C01819=1081.465,156.969,428.718,174.663,22.838,153.849
C01820=1081.471,157.219,428.696,174.666,22.840,153.849
C01821=1081.476,157.468,428.675,174.667,22.842,153.849
C01822=1081.482,157.716,428.654,174.670,22.844,153.849
C01823=1081.488,157.966,428.633,174.672,22.846,153.850
C01824=1081.493,158.215,428.611,174.674,22.848,153.850
C01825=1081.499,158.463,428.590,174.676,22.850,153.850
C01826=1081.505,158.713,428.569,174.678,22.852,153.850
C01827=1081.510,158.962,428.548,174.680,22.854,153.850
C01828=1081.517,159.241,428.524,174.683,22.857,153.850
C01829=1081.523,159.522,428.500,174.685,22.859,153.850
C01830=1081.529,159.801,428.476,174.687,22.861,153.850
C01831=1081.535,160.081,428.452,174.690,22.863,153.851
C01832=1081.541,160.330,428.430,174.692,22.866,153.851
C01833=1081.546,160.579,428.409,174.694,22.868,153.851
C01834=1081.552,160.829,428.388,174.697,22.870,153.851
C01835=1081.558,161.077,428.366,174.698,22.872,153.851
C01836=1081.564,161.327,428.345,174.701,22.874,153.851
C01837=1081.569,161.575,428.323,174.703,22.876,153.851
C01838=1081.574,161.824,428.302,174.705,22.879,153.851
C01839=1081.580,162.074,428.281,174.707,22.880,153.852
C01840=1081.585,162.323,428.259,174.709,22.883,153.852
C01841=1081.590,162.571,428.238,174.711,22.885,153.852
C01842=1081.596,162.821,428.215,174.714,22.887,153.852
C01843=1081.601,163.069,428.194,174.716,22.889,153.852
C01844=1081.608,163.318,428.172,174.718,22.891,153.852
C01845=1081.612,163.567,428.151,174.720,22.893,153.852
C01846=1081.619,163.816,428.129,174.722,22.895,153.853
C01847=1081.623,164.066,428.108,174.725,22.898,153.853
C01848=1081.629,164.314,428.086,174.727,22.900,153.853
C01849=1081.634,164.564,428.064,174.728,22.902,153.853
C01850=1081.640,164.812,428.043,174.731,22.904,153.853
C01851=1081.645,165.062,428.021,174.733,22.906,153.853
C01852=1081.651,165.310,427.999,174.735,22.908,153.853
C01853=1081.656,165.560,427.977,174.738,22.910,153.853
C01854=1081.662,165.808,427.956,174.739,22.912,153.854
C01855=1081.667,166.058,427.934,174.742,22.915,153.854
C01856=1081.673,166.306,427.912,174.744,22.917,153.854
C01857=1081.677,166.555,427.891,174.746,22.919,153.854
C01858=1081.684,166.804,427.869,174.749,22.921,153.854
C01859=1081.688,167.053,427.847,174.750,22.923,153.854
C01860=1081.695,167.302,427.825,174.752,22.925,153.854
C01861=1081.699,167.551,427.804,174.755,22.927,153.855
C01862=1081.706,167.800,427.782,174.757,22.930,153.855
C01863=1081.710,168.049,427.760,174.759,22.932,153.855
C01864=1081.716,168.298,427.738,174.761,22.933,153.855
C01865=1081.721,168.547,427.717,174.763,22.935,153.855
C01866=1081.728,168.796,427.694,174.766,22.938,153.855
C01867=1081.733,169.045,427.672,174.768,22.940,153.855
C01868=1081.739,169.294,427.651,174.770,22.942,153.855
C01869=1081.744,169.543,427.629,174.773,22.944,153.855
C01870=1081.749,169.792,427.607,174.774,22.946,153.856
C01871=1081.755,170.041,427.585,174.777,22.948,153.856
C01872=1081.760,170.290,427.563,174.779,22.950,153.856
C01873=1081.766,170.539,427.541,174.781,22.953,153.856
C01874=1081.771,170.788,427.519,174.784,22.954,153.856
C01875=1081.777,171.037,427.497,174.786,22.957,153.856
C01876=1081.783,171.286,427.475,174.788,22.959,153.856
C01877=1081.788,171.535,427.454,174.790,22.961,153.856
C01878=1081.794,171.784,427.431,174.792,22.963,153.856
C01879=1081.799,172.032,427.409,174.795,22.965,153.857
C01880=1081.805,172.282,427.387,174.797,22.967,153.857
C01881=1081.811,172.531,427.365,174.799,22.969,153.857
C01882=1081.816,172.779,427.343,174.801,22.971,153.857
C01883=1081.822,173.029,427.321,174.803,22.973,153.857
C01884=1081.827,173.278,427.299,174.806,22.975,153.857
C01885=1081.833,173.527,427.277,174.808,22.978,153.857
C01886=1081.839,173.776,427.254,174.810,22.979,153.857
C01887=1081.844,174.024,427.233,174.813,22.982,153.858
C01888=1081.850,174.274,427.211,174.815,22.984,153.858
C01889=1081.855,174.522,427.188,174.817,22.985,153.858
C01890=1081.861,174.771,427.167,174.819,22.988,153.858
C01891=1081.866,175.020,427.145,174.821,22.990,153.858
C01892=1081.873,175.300,427.119,174.824,22.992,153.858
C01893=1081.879,175.580,427.094,174.827,22.995,153.858
C01894=1081.886,175.859,427.069,174.829,22.997,153.858
C01895=1081.892,176.138,427.045,174.832,22.999,153.858
C01896=1081.897,176.387,427.023,174.834,23.001,153.859
C01897=1081.903,176.636,427.000,174.836,23.003,153.859
C01898=1081.909,176.885,426.978,174.839,23.005,153.859
C01899=1081.914,177.134,426.956,174.841,23.007,153.859
C01900=1081.920,177.383,426.933,174.843,23.009,153.859
C01901=1081.926,177.632,426.911,174.845,23.011,153.859
C01902=1081.932,177.881,426.889,174.847,23.013,153.859
C01903=1081.937,178.129,426.866,174.850,23.016,153.859
C01904=1081.942,178.379,426.844,174.852,23.017,153.859
C01905=1081.949,178.627,426.822,174.855,23.020,153.860
C01906=1081.954,178.877,426.799,174.857,23.022,153.860
C01907=1081.959,179.125,426.777,174.860,23.024,153.860
C01908=1081.965,179.374,426.755,174.862,23.026,153.860
C01909=1081.971,179.623,426.732,174.864,23.028,153.860
C01910=1081.977,179.873,426.710,174.866,23.029,153.860
C01911=1081.982,180.121,426.688,174.868,23.032,153.860
C01912=1081.988,180.370,426.666,174.871,23.033,153.860
C01913=1081.994,180.619,426.643,174.873,23.036,153.860
C01914=1081.999,180.868,426.620,174.875,23.037,153.860
C01915=1082.005,181.117,426.598,174.878,23.040,153.860
C01916=1082.011,181.366,426.575,174.880,23.042,153.861
C01917=1082.016,181.615,426.554,174.883,23.044,153.861
C01918=1082.023,181.863,426.531,174.885,23.046,153.861
C01919=1082.028,182.112,426.508,174.887,23.048,153.861
C01920=1082.034,182.362,426.486,174.890,23.050,153.861
C01921=1082.039,182.611,426.463,174.891,23.051,153.861
C01922=1082.046,182.859,426.441,174.894,23.054,153.861
C01923=1082.052,183.108,426.418,174.896,23.056,153.861
C01924=1082.056,183.357,426.396,174.899,23.058,153.861
C01925=1082.062,183.606,426.373,174.901,23.060,153.861
C01926=1082.068,183.855,426.350,174.903,23.062,153.861
C01927=1082.074,184.104,426.328,174.906,23.064,153.862
C01928=1082.080,184.353,426.305,174.908,23.066,153.862
C01929=1082.086,184.602,426.282,174.911,23.068,153.862
C01930=1082.091,184.851,426.260,174.913,23.070,153.862
C01931=1082.097,185.100,426.237,174.915,23.072,153.862
C01932=1082.102,185.348,426.215,174.918,23.074,153.862
C01933=1082.108,185.597,426.192,174.920,23.077,153.862
C01934=1082.113,185.846,426.169,174.923,23.078,153.862
C01935=1082.119,186.095,426.146,174.925,23.081,153.862
C01936=1082.125,186.344,426.123,174.927,23.083,153.862
C01937=1082.130,186.593,426.101,174.929,23.085,153.863
C01938=1082.135,186.842,426.078,174.931,23.087,153.863
C01939=1082.140,187.091,426.055,174.934,23.089,153.863
C01940=1082.146,187.340,426.032,174.936,23.091,153.863
C01941=1082.152,187.589,426.009,174.938,23.093,153.863
C01942=1082.157,187.837,425.986,174.941,23.095,153.863
C01943=1082.163,188.086,425.963,174.943,23.097,153.863
C01944=1082.168,188.335,425.940,174.945,23.099,153.863
C01945=1082.173,188.584,425.917,174.948,23.102,153.864
C01946=1082.179,188.833,425.894,174.950,23.104,153.864
C01947=1082.185,189.082,425.871,174.953,23.106,153.864
C01948=1082.190,189.331,425.848,174.955,23.108,153.864
C01949=1082.196,189.579,425.825,174.957,23.110,153.864
C01950=1082.201,189.828,425.802,174.960,23.112,153.864
C01951=1082.206,190.077,425.779,174.962,23.114,153.864
C01952=1082.212,190.326,425.756,174.964,23.117,153.864
C01953=1082.218,190.575,425.733,174.967,23.119,153.864
C01954=1082.224,190.824,425.710,174.969,23.121,153.864
C01955=1082.229,191.073,425.686,174.972,23.123,153.865
C01956=1082.235,191.352,425.661,174.974,23.125,153.865
C01957=1082.241,191.632,425.635,174.977,23.128,153.865
C01958=1082.247,191.910,425.609,174.980,23.130,153.865
C01959=1082.253,192.189,425.583,174.982,23.132,153.865
C01960=1082.259,192.438,425.560,174.984,23.134,153.865
C01961=1082.264,192.687,425.537,174.987,23.136,153.865
C01962=1082.270,192.936,425.514,174.989,23.139,153.865
C01963=1082.275,193.185,425.491,174.992,23.140,153.865
C01964=1082.281,193.434,425.468,174.994,23.143,153.866
C01965=1082.287,193.682,425.444,174.996,23.145,153.866
C01966=1082.293,193.931,425.421,174.999,23.147,153.866
C01967=1082.298,194.180,425.398,175.001,23.149,153.866
C01968=1082.303,194.429,425.375,175.003,23.151,153.866
C01969=1082.309,194.678,425.352,175.006,23.153,153.866
C01970=1082.315,194.926,425.328,175.008,23.155,153.866
C01971=1082.320,195.176,425.304,175.012,23.158,153.866
C01972=1082.326,195.424,425.281,175.014,23.159,153.866
C01973=1082.331,195.673,425.259,175.016,23.162,153.867
C01974=1082.337,195.922,425.234,175.019,23.164,153.867
C01975=1082.343,196.171,425.211,175.021,23.166,153.867
C01976=1082.348,196.420,425.188,175.024,23.168,153.867
C01977=1082.354,196.669,425.165,175.026,23.170,153.867
C01978=1082.359,196.917,425.141,175.028,23.172,153.867
C01979=1082.365,197.166,425.118,175.031,23.174,153.867
C01980=1082.371,197.415,425.095,175.033,23.177,153.867
C01981=1082.376,197.664,425.071,175.036,23.178,153.867
C01982=1082.382,197.913,425.048,175.038,23.181,153.867
C01983=1082.388,198.162,425.025,175.040,23.182,153.867
C01984=1082.393,198.411,425.001,175.043,23.185,153.868
C01985=1082.399,198.660,424.978,175.045,23.187,153.868
C01986=1082.405,198.908,424.954,175.048,23.189,153.868
C01987=1082.410,199.157,424.930,175.050,23.191,153.868
C01988=1082.416,199.406,424.907,175.053,23.193,153.868
C01989=1082.421,199.655,424.883,175.055,23.195,153.868
C01990=1082.427,199.903,424.860,175.057,23.197,153.868
C01991=1082.434,200.152,424.836,175.060,23.199,153.868
C01992=1082.439,200.402,424.813,175.062,23.201,153.868
C01993=1082.445,200.650,424.789,175.065,23.203,153.868
C01994=1082.450,200.899,424.766,175.068,23.205,153.869
C01995=1082.456,201.147,424.742,175.070,23.208,153.869
C01996=1082.461,201.396,424.719,175.073,23.209,153.869
C01997=1082.467,201.645,424.695,175.075,23.212,153.869
C01998=1082.473,201.895,424.671,175.078,23.213,153.869
C01999=1082.479,202.143,424.648,175.080,23.216,153.869
C02000=1082.484,202.392,424.624,175.082,23.218,153.869
C02001=1082.490,202.640,424.600,175.085,23.220,153.869
C02002=1082.495,202.889,424.577,175.087,23.222,153.869
C02003=1082.501,203.138,424.553,175.089,23.224,153.869
C02004=1082.507,203.387,424.529,175.092,23.226,153.869
C02005=1082.512,203.636,424.505,175.094,23.228,153.870
C02006=1082.518,203.885,424.481,175.098,23.231,153.870
C02007=1082.523,204.134,424.458,175.100,23.233,153.870
C02008=1082.529,204.382,424.434,175.102,23.235,153.870
C02009=1082.534,204.631,424.410,175.105,23.237,153.870
C02010=1082.539,204.880,424.386,175.107,23.239,153.870
C02011=1082.546,205.129,424.362,175.110,23.241,153.870
C02012=1082.551,205.377,424.338,175.112,23.243,153.870
C02013=1082.556,205.627,424.315,175.114,23.246,153.871
C02014=1082.562,205.875,424.291,175.117,23.247,153.871
C02015=1082.568,206.123,424.267,175.120,23.250,153.871
C02016=1082.573,206.373,424.242,175.122,23.252,153.871
C02017=1082.579,206.622,424.219,175.125,23.254,153.871
C02018=1082.585,206.870,424.195,175.127,23.256,153.871
C02019=1082.590,207.119,424.171,175.130,23.258,153.871
C02020=1082.613,208.150,424.072,175.222,23.307,153.869
C02021=1082.623,208.544,424.032,175.226,23.312,153.869
C02022=1082.632,208.938,423.993,175.229,23.317,153.870
C02023=1082.640,209.332,423.955,175.233,23.321,153.870
C02024=1082.649,209.727,423.916,175.236,23.326,153.871
C02025=1082.655,209.975,423.891,175.239,23.330,153.871
C02026=1082.661,210.224,423.866,175.241,23.332,153.871
C02027=1082.666,210.472,423.842,175.243,23.336,153.872
C02028=1082.672,210.722,423.818,175.246,23.339,153.872
C02029=1082.677,210.970,423.793,175.249,23.342,153.872
C02030=1082.683,211.219,423.768,175.251,23.345,153.873
C02031=1082.689,211.468,423.744,175.254,23.348,153.873
C02032=1082.695,211.716,423.718,175.256,23.351,153.873
C02033=1082.700,211.965,423.694,175.258,23.354,153.874
C02034=1082.705,212.213,423.670,175.261,23.357,153.874
C02035=1082.712,212.462,423.644,175.263,23.360,153.874
C02036=1082.717,212.711,423.620,175.265,23.363,153.875
C02037=1082.723,212.960,423.596,175.268,23.366,153.875
C02038=1082.728,213.208,423.571,175.270,23.370,153.875
C02039=1082.734,213.457,423.546,175.272,23.372,153.876
C02040=1082.740,213.705,423.521,175.275,23.376,153.876
C02041=1082.746,213.955,423.496,175.277,23.379,153.876
C02042=1082.750,214.203,423.472,175.279,23.382,153.877
C02043=1082.757,214.452,423.446,175.283,23.385,153.877
C02044=1082.762,214.701,423.422,175.285,23.388,153.877
C02045=1082.768,214.949,423.397,175.287,23.391,153.878
C02046=1082.773,215.198,423.372,175.290,23.394,153.878
C02047=1082.779,215.447,423.346,175.292,23.398,153.878
C02048=1082.784,215.695,423.322,175.294,23.400,153.879
C02049=1082.790,215.944,423.297,175.297,23.404,153.879
C02050=1082.796,216.193,423.272,175.299,23.407,153.879
C02051=1082.802,216.441,423.247,175.301,23.410,153.879
C02052=1082.807,216.690,423.221,175.304,23.413,153.880
C02053=1082.813,216.939,423.197,175.306,23.416,153.880
C02054=1082.819,217.188,423.172,175.309,23.419,153.880
C02055=1082.824,217.436,423.147,175.311,23.422,153.881
C02056=1082.830,217.685,423.122,175.314,23.425,153.881
C02057=1082.836,217.934,423.096,175.316,23.428,153.881
C02058=1082.841,218.182,423.072,175.319,23.432,153.882
C02059=1082.847,218.431,423.047,175.321,23.434,153.882
C02060=1082.852,218.680,423.022,175.323,23.438,153.882
C02061=1082.858,218.929,422.996,175.326,23.441,153.883
C02062=1082.864,219.177,422.971,175.328,23.443,153.883
C02063=1082.870,219.425,422.946,175.331,23.447,153.883
C02064=1082.875,219.675,422.921,175.333,23.450,153.884
C02065=1082.881,219.924,422.896,175.336,23.453,153.884
C02066=1082.887,220.172,422.871,175.338,23.456,153.884
C02067=1082.893,220.421,422.846,175.341,23.459,153.885
C02068=1082.898,220.670,422.820,175.343,23.462,153.885
C02069=1082.904,220.918,422.795,175.346,23.465,153.885
C02070=1082.910,221.166,422.770,175.348,23.468,153.886
C02071=1082.916,221.415,422.744,175.351,23.471,153.886
C02072=1082.921,221.664,422.720,175.353,23.475,153.886
C02073=1082.930,222.062,422.679,175.357,23.479,153.887
C02074=1082.940,222.461,422.638,175.361,23.485,153.887
C02075=1082.948,222.859,422.597,175.365,23.489,153.888
C02076=1082.957,223.256,422.556,175.369,23.495,153.888
C02077=1082.963,223.504,422.531,175.371,23.497,153.889
C02078=1082.968,223.754,422.506,175.373,23.501,153.889
C02079=1082.974,224.003,422.481,175.376,23.504,153.889
C02080=1082.980,224.252,422.455,175.379,23.507,153.890
C02081=1082.985,224.499,422.430,175.382,23.510,153.890
C02082=1082.991,224.748,422.404,175.384,23.513,153.890
C02083=1082.997,224.997,422.378,175.386,23.516,153.891
C02084=1083.002,225.245,422.353,175.389,23.519,153.891
C02085=1083.007,225.494,422.327,175.391,23.522,153.891
C02086=1083.013,225.743,422.302,175.394,23.526,153.892
C02087=1083.019,225.992,422.276,175.396,23.528,153.892
C02088=1083.025,226.240,422.251,175.398,23.532,153.892
C02089=1083.030,226.489,422.225,175.401,23.535,153.893
C02090=1083.036,226.738,422.199,175.403,23.538,153.893
C02091=1083.042,226.987,422.173,175.406,23.541,153.893
C02092=1083.048,227.234,422.148,175.409,23.544,153.893
C02093=1083.053,227.483,422.122,175.411,23.547,153.894
C02094=1083.059,227.732,422.096,175.414,23.550,153.894
C02095=1083.065,227.981,422.071,175.416,23.553,153.894
C02096=1083.070,228.230,422.045,175.419,23.557,153.895
C02097=1083.076,228.478,422.019,175.421,23.560,153.895
C02098=1083.081,228.727,421.994,175.424,23.563,153.895
C02099=1083.088,228.975,421.968,175.426,23.566,153.896
C02100=1083.093,229.224,421.942,175.428,23.569,153.896
C02101=1083.099,229.473,421.916,175.431,23.572,153.896
C02102=1083.105,229.721,421.891,175.433,23.575,153.897
C02103=1083.110,229.970,421.865,175.437,23.578,153.897
C02104=1083.116,230.218,421.838,175.439,23.581,153.897
C02105=1083.122,230.467,421.813,175.442,23.585,153.898
C02106=1083.127,230.715,421.787,175.444,23.587,153.898
C02107=1083.133,230.964,421.760,175.446,23.591,153.898
C02108=1083.139,231.213,421.734,175.449,23.594,153.899
C02109=1083.145,231.462,421.709,175.451,23.597,153.899
C02110=1083.150,231.710,421.684,175.454,23.600,153.899
C02111=1083.155,231.958,421.657,175.456,23.603,153.900
C02112=1083.161,232.207,421.631,175.459,23.606,153.900
C02113=1083.167,232.456,421.606,175.461,23.609,153.900
C02114=1083.173,232.704,421.579,175.464,23.613,153.901
C02115=1083.178,232.953,421.553,175.467,23.616,153.901
C02116=1083.184,233.201,421.526,175.469,23.619,153.901
C02117=1083.190,233.450,421.500,175.472,23.622,153.902
C02118=1083.195,233.699,421.475,175.474,23.625,153.902
C02119=1083.201,233.947,421.449,175.477,23.628,153.902
C02120=1083.206,234.196,421.423,175.479,23.631,153.903
C02121=1083.212,234.444,421.396,175.482,23.635,153.903
C02122=1083.218,234.693,421.370,175.484,23.637,153.903
C02123=1083.223,234.941,421.344,175.487,23.641,153.904
C02124=1083.229,235.190,421.318,175.489,23.644,153.904
C02125=1083.238,235.580,421.276,175.494,23.649,153.905
C02126=1083.246,235.969,421.235,175.497,23.654,153.905
C02127=1083.255,236.359,421.194,175.501,23.658,153.905
C02128=1083.264,236.748,421.153,175.506,23.664,153.906
C02129=1083.269,236.997,421.126,175.508,23.666,153.906
C02130=1083.275,237.246,421.101,175.511,23.670,153.907
C02131=1083.281,237.494,421.074,175.513,23.673,153.907
C02132=1083.287,237.742,421.047,175.516,23.676,153.907
C02133=1083.292,237.991,421.021,175.518,23.679,153.908
C02134=1083.298,238.240,420.995,175.521,23.682,153.908
C02135=1083.304,238.488,420.968,175.523,23.686,153.908
C02136=1083.310,238.737,420.943,175.526,23.689,153.909
C02137=1083.316,238.985,420.916,175.528,23.692,153.909
C02138=1083.321,239.233,420.889,175.531,23.695,153.909
C02139=1083.327,239.482,420.863,175.534,23.698,153.910
C02140=1083.333,239.731,420.837,175.537,23.701,153.910
C02141=1083.338,239.980,420.809,175.539,23.704,153.910
C02142=1083.344,240.228,420.783,175.542,23.708,153.911
C02143=1083.350,240.477,420.756,175.544,23.710,153.911
C02144=1083.355,240.726,420.730,175.547,23.714,153.911
C02145=1083.361,240.974,420.703,175.549,23.717,153.912
C02146=1083.367,241.223,420.677,175.552,23.720,153.912
C02147=1083.372,241.471,420.650,175.554,23.723,153.912
C02148=1083.378,241.719,420.623,175.557,23.726,153.913
C02149=1083.384,241.968,420.597,175.559,23.730,153.913
C02150=1083.390,242.217,420.571,175.562,23.733,153.913
C02151=1083.395,242.465,420.544,175.565,23.735,153.914
C02152=1083.401,242.713,420.517,175.568,23.739,153.914
C02153=1083.407,242.962,420.491,175.570,23.742,153.914
C02154=1083.412,243.210,420.464,175.573,23.745,153.915
C02155=1083.418,243.459,420.437,175.575,23.748,153.915
C02156=1083.424,243.708,420.410,175.578,23.752,153.915
C02157=1083.430,243.956,420.383,175.580,23.754,153.916
C02158=1083.435,244.205,420.356,175.583,23.758,153.916
C02159=1083.441,244.453,420.329,175.585,23.761,153.916
C02160=1083.446,244.702,420.303,175.588,23.764,153.917
C02161=1083.451,244.950,420.276,175.591,23.768,153.917
C02162=1083.457,245.199,420.249,175.593,23.771,153.917
C02163=1083.463,245.447,420.222,175.597,23.774,153.918
C02164=1083.469,245.695,420.196,175.599,23.777,153.918
C02165=1083.474,245.945,420.168,175.602,23.780,153.918
C02166=1083.480,246.193,420.141,175.604,23.783,153.919
C02167=1083.486,246.441,420.115,175.607,23.787,153.919
C02168=1083.491,246.690,420.087,175.609,23.790,153.919
C02169=1083.497,246.938,420.061,175.612,23.793,153.920
C02170=1083.503,247.186,420.033,175.614,23.796,153.920
C02171=1083.508,247.435,420.006,175.617,23.799,153.920
C02172=1083.514,247.684,419.979,175.619,23.802,153.921
C02173=1083.519,247.933,419.952,175.622,23.806,153.921
C02174=1083.525,248.181,419.925,175.625,23.809,153.921
C02175=1083.530,248.430,419.898,175.627,23.812,153.922
C02176=1083.536,248.677,419.871,175.631,23.815,153.922
C02177=1083.544,249.061,419.829,175.634,23.821,153.923
C02178=1083.553,249.443,419.787,175.639,23.825,153.923
C02179=1083.562,249.826,419.745,175.642,23.830,153.924
C02180=1083.570,250.208,419.703,175.647,23.835,153.924
C02181=1083.576,250.457,419.676,175.649,23.839,153.925
C02182=1083.581,250.705,419.649,175.652,23.842,153.925
C02183=1083.587,250.953,419.621,175.654,23.845,153.925
C02184=1083.593,251.203,419.594,175.657,23.849,153.926
C02185=1083.598,251.451,419.567,175.659,23.851,153.926
C02186=1083.604,251.699,419.539,175.662,23.855,153.926
C02187=1083.609,251.948,419.512,175.665,23.858,153.927
C02188=1083.616,252.197,419.485,175.667,23.861,153.927
C02189=1083.621,252.445,419.457,175.670,23.865,153.927
C02190=1083.627,252.693,419.430,175.673,23.868,153.928
C02191=1083.632,252.941,419.402,175.676,23.871,153.928
C02192=1083.638,253.190,419.375,175.679,23.874,153.928
C02193=1083.644,253.438,419.347,175.681,23.877,153.929
C02194=1083.649,253.687,419.320,175.684,23.881,153.929
C02195=1083.655,253.935,419.293,175.686,23.884,153.930
C02196=1083.660,254.184,419.265,175.689,23.887,153.930
C02197=1083.667,254.432,419.238,175.691,23.890,153.930
C02198=1083.672,254.680,419.211,175.694,23.894,153.931
C02199=1083.678,254.929,419.182,175.697,23.897,153.931
C02200=1083.683,255.178,419.156,175.699,23.900,153.931
C02201=1083.689,255.426,419.128,175.702,23.903,153.932
C02202=1083.695,255.674,419.099,175.704,23.906,153.932
C02203=1083.700,255.923,419.073,175.708,23.909,153.932
C02204=1083.706,256.171,419.045,175.711,23.913,153.933
C02205=1083.712,256.420,419.018,175.713,23.916,153.933
C02206=1083.717,256.668,418.990,175.716,23.919,153.933
C02207=1083.723,256.916,418.962,175.718,23.922,153.934
C02208=1083.729,257.165,418.935,175.721,23.926,153.934
C02209=1083.734,257.413,418.907,175.724,23.929,153.934
C02210=1083.740,257.662,418.878,175.726,23.932,153.935
C02211=1083.747,257.910,418.851,175.729,23.936,153.935
C02212=1083.752,258.158,418.824,175.732,23.939,153.935
C02213=1083.757,258.407,418.796,175.734,23.942,153.936
C02214=1083.764,258.655,418.768,175.737,23.945,153.936
C02215=1083.770,258.904,418.740,175.739,23.948,153.936
C02216=1083.775,259.152,418.713,175.743,23.951,153.937
C02217=1083.780,259.401,418.684,175.746,23.955,153.937
C02218=1083.787,259.649,418.657,175.748,23.958,153.937
C02219=1083.793,259.897,418.629,175.751,23.961,153.938
C02220=1083.798,260.145,418.601,175.754,23.964,153.938
C02221=1083.804,260.393,418.573,175.756,23.967,153.938
C02222=1083.810,260.643,418.546,175.759,23.971,153.939
C02223=1083.815,260.891,418.518,175.761,23.974,153.939
C02224=1083.821,261.139,418.489,175.764,23.977,153.939
C02225=1083.827,261.387,418.462,175.767,23.980,153.940
C02226=1083.833,261.636,418.434,175.770,23.983,153.940
C02227=1083.838,261.884,418.406,175.772,23.987,153.941
C02228=1083.844,262.133,418.377,175.776,23.990,153.941
C02229=1083.853,262.512,418.335,175.779,23.995,153.941
C02230=1083.863,262.892,418.292,175.784,24.000,153.942
C02231=1083.871,263.272,418.249,175.788,24.004,153.942
C02232=1083.880,263.652,418.206,175.792,24.010,153.943
C02233=1083.886,263.901,418.178,175.795,24.013,153.943
C02234=1083.892,264.149,418.150,175.797,24.016,153.944
C02235=1083.897,264.398,418.122,175.800,24.019,153.944
C02236=1083.903,264.646,418.094,175.803,24.023,153.944
C02237=1083.909,264.895,418.065,175.805,24.026,153.945
C02238=1083.914,265.142,418.037,175.808,24.029,153.945
C02239=1083.920,265.391,418.008,175.812,24.032,153.945
C02240=1083.926,265.639,417.980,175.814,24.036,153.946
C02241=1083.932,265.888,417.952,175.817,24.039,153.946
C02242=1083.937,266.136,417.924,175.820,24.042,153.946
C02243=1083.943,266.384,417.896,175.822,24.046,153.947
C02244=1083.949,266.632,417.867,175.825,24.049,153.947
C02245=1083.954,266.881,417.839,175.828,24.052,153.948
C02246=1083.960,267.129,417.811,175.830,24.055,153.948
C02247=1083.966,267.377,417.782,175.833,24.059,153.948
C02248=1083.972,267.626,417.753,175.836,24.062,153.949
C02249=1083.977,267.874,417.725,175.838,24.065,153.949
C02250=1083.983,268.122,417.697,175.841,24.069,153.949
C02251=1083.989,268.370,417.669,175.844,24.072,153.950
C02252=1083.994,268.619,417.640,175.846,24.075,153.950
C02253=1084.000,268.868,417.611,175.849,24.079,153.951
C02254=1084.005,269.116,417.583,175.853,24.082,153.951
C02255=1084.012,269.364,417.554,175.856,24.085,153.951
C02256=1084.018,269.613,417.526,175.858,24.089,153.952
C02257=1084.023,269.860,417.497,175.861,24.092,153.952
C02258=1084.029,270.109,417.469,175.864,24.095,153.952
C02259=1084.034,270.357,417.440,175.866,24.098,153.953
C02260=1084.040,270.605,417.411,175.869,24.102,153.953
C02261=1084.046,270.854,417.383,175.872,24.105,153.953
C02262=1084.052,271.101,417.354,175.874,24.108,153.954
C02263=1084.058,271.350,417.326,175.877,24.112,153.954
C02264=1084.063,271.599,417.296,175.880,24.115,153.955
C02265=1084.068,271.847,417.268,175.883,24.119,153.955
C02266=1084.075,272.095,417.239,175.885,24.122,153.955
C02267=1084.081,272.344,417.211,175.888,24.125,153.956
C02268=1084.086,272.591,417.182,175.891,24.129,153.956
C02269=1084.092,272.840,417.153,175.893,24.132,153.956
C02270=1084.098,273.088,417.124,175.896,24.135,153.957
C02271=1084.103,273.336,417.096,175.899,24.139,153.957
C02272=1084.109,273.585,417.067,175.902,24.142,153.958
C02273=1084.115,273.833,417.038,175.905,24.145,153.958
C02274=1084.121,274.082,417.009,175.908,24.149,153.958
C02275=1084.126,274.329,416.980,175.911,24.152,153.959
C02276=1084.132,274.577,416.951,175.913,24.155,153.959
C02277=1084.137,274.827,416.922,175.916,24.159,153.960
C02278=1084.143,275.074,416.894,175.919,24.162,153.960
C02279=1084.149,275.322,416.864,175.922,24.166,153.960
C02280=1084.154,275.571,416.836,175.924,24.169,153.961
C02281=1084.163,275.954,416.790,175.928,24.174,153.961
C02282=1084.172,276.337,416.746,175.933,24.179,153.962
C02283=1084.181,276.719,416.701,175.937,24.185,153.962
C02284=1084.190,277.102,416.656,175.941,24.190,153.963
C02285=1084.195,277.350,416.628,175.944,24.193,153.963
C02286=1084.201,277.599,416.598,175.947,24.196,153.964
C02287=1084.207,277.847,416.569,175.950,24.200,153.964
C02288=1084.213,278.095,416.539,175.952,24.203,153.965
C02289=1084.219,278.343,416.510,175.955,24.207,153.965
C02290=1084.224,278.591,416.481,175.958,24.210,153.965
C02291=1084.230,278.839,416.452,175.961,24.214,153.966
C02292=1084.236,279.088,416.422,175.964,24.217,153.966
C02293=1084.241,279.336,416.394,175.967,24.220,153.966
C02294=1084.247,279.585,416.364,175.970,24.224,153.967
C02295=1084.253,279.832,416.336,175.973,24.227,153.967
C02296=1084.258,280.081,416.306,175.976,24.231,153.968
C02297=1084.264,280.329,416.277,175.978,24.234,153.968
C02298=1084.270,280.577,416.247,175.981,24.238,153.968
C02299=1084.276,280.825,416.218,175.984,24.241,153.969
C02300=1084.282,281.074,416.189,175.987,24.244,153.969
C02301=1084.287,281.322,416.159,175.989,24.247,153.970
C02302=1084.293,281.569,416.130,175.992,24.251,153.970
C02303=1084.299,281.818,416.100,175.995,24.254,153.970
C02304=1084.304,282.066,416.071,175.998,24.258,153.971
C02305=1084.310,282.314,416.041,176.001,24.262,153.971
C02306=1084.316,282.563,416.012,176.003,24.265,153.972
C02307=1084.321,282.811,415.982,176.006,24.268,153.972
C02308=1084.326,283.059,415.953,176.009,24.272,153.972
C02309=1084.333,283.307,415.924,176.012,24.275,153.973
C02310=1084.338,283.555,415.894,176.014,24.279,153.973
C02311=1084.344,283.803,415.864,176.017,24.282,153.974
C02312=1084.349,284.052,415.834,176.020,24.286,153.974
C02313=1084.356,284.300,415.805,176.023,24.289,153.974
C02314=1084.361,284.547,415.775,176.026,24.293,153.975
C02315=1084.367,284.796,415.745,176.028,24.296,153.975
C02316=1084.372,285.044,415.716,176.031,24.300,153.976
C02317=1084.379,285.293,415.687,176.034,24.303,153.976
C02318=1084.385,285.540,415.656,176.037,24.307,153.976
C02319=1084.389,285.788,415.627,176.040,24.310,153.977
C02320=1084.395,286.037,415.597,176.042,24.313,153.977
C02321=1084.402,286.284,415.568,176.045,24.317,153.978
C02322=1084.407,286.532,415.538,176.048,24.321,153.978
C02323=1084.413,286.781,415.508,176.052,24.324,153.979
C02324=1084.418,287.029,415.478,176.055,24.328,153.979
C02325=1084.424,287.277,415.448,176.058,24.331,153.979
C02326=1084.430,287.525,415.419,176.060,24.334,153.980
C02327=1084.436,287.773,415.389,176.063,24.338,153.980
C02328=1084.441,288.022,415.359,176.066,24.342,153.981
C02329=1084.447,288.269,415.329,176.069,24.345,153.981
C02330=1084.453,288.518,415.299,176.072,24.349,153.981
C02331=1084.459,288.766,415.269,176.075,24.352,153.982
C02332=1084.465,289.014,415.240,176.077,24.355,153.982
C02333=1084.474,289.407,415.191,176.081,24.361,153.983
C02334=1084.483,289.799,415.145,176.087,24.367,153.984
C02335=1084.492,290.191,415.097,176.091,24.372,153.984
C02336=1084.501,290.584,415.050,176.096,24.378,153.985
C02337=1084.507,290.832,415.019,176.099,24.382,153.985
C02338=1084.513,291.080,414.989,176.101,24.385,153.986
C02339=1084.518,291.328,414.959,176.104,24.388,153.986
C02340=1084.525,291.576,414.929,176.107,24.392,153.987
C02341=1084.531,291.824,414.898,176.110,24.396,153.987
C02342=1084.536,292.073,414.869,176.113,24.399,153.987
C02343=1084.542,292.321,414.838,176.116,24.403,153.988
C02344=1084.548,292.568,414.808,176.119,24.406,153.988
C02345=1084.553,292.817,414.778,176.121,24.410,153.989
C02346=1084.558,293.065,414.747,176.124,24.413,153.989
C02347=1084.564,293.313,414.717,176.127,24.417,153.990
C02348=1084.570,293.561,414.687,176.130,24.421,153.990
C02349=1084.576,293.808,414.656,176.133,24.424,153.990
C02350=1084.581,294.057,414.627,176.136,24.428,153.991
C02351=1084.588,294.305,414.596,176.139,24.431,153.991
C02352=1084.594,294.553,414.566,176.141,24.435,153.992
C02353=1084.599,294.801,414.535,176.144,24.439,153.992
C02354=1084.605,295.049,414.505,176.147,24.442,153.993
C02355=1084.611,295.297,414.475,176.150,24.446,153.993
C02356=1084.616,295.545,414.444,176.153,24.449,153.993
C02357=1084.622,295.794,414.414,176.156,24.453,153.994
C02358=1084.628,296.042,414.383,176.159,24.457,153.994
C02359=1084.634,296.290,414.353,176.162,24.460,153.995
C02360=1084.640,296.537,414.323,176.165,24.464,153.995
C02361=1084.645,296.786,414.292,176.167,24.468,153.996
C02362=1084.650,297.033,414.261,176.170,24.471,153.996
C02363=1084.657,297.282,414.231,176.173,24.475,153.997
C02364=1084.663,297.530,414.200,176.176,24.479,153.997
C02365=1084.669,297.778,414.170,176.179,24.482,153.997
C02366=1084.674,298.026,414.139,176.182,24.486,153.998
C02367=1084.679,298.273,414.109,176.185,24.490,153.998
C02368=1084.685,298.522,414.078,176.188,24.493,153.999
C02369=1084.691,298.770,414.046,176.191,24.497,153.999
C02370=1084.697,299.017,414.016,176.194,24.501,154.000
C02371=1084.702,299.265,413.985,176.196,24.505,154.000
C02372=1084.708,299.513,413.955,176.199,24.508,154.001
C02373=1084.713,299.761,413.924,176.202,24.512,154.001
C02374=1084.719,300.009,413.893,176.204,24.516,154.002
C02375=1084.725,300.257,413.861,176.208,24.519,154.002
C02376=1084.731,300.505,413.831,176.210,24.523,154.003
C02377=1084.736,300.753,413.800,176.213,24.527,154.003
C02378=1084.742,301.001,413.770,176.216,24.531,154.004
C02379=1084.747,301.249,413.739,176.219,24.534,154.004
C02380=1084.753,301.497,413.707,176.222,24.538,154.005
C02381=1084.758,301.745,413.676,176.225,24.542,154.005
C02382=1084.764,301.993,413.646,176.228,24.546,154.005
C02383=1084.770,302.241,413.614,176.231,24.549,154.006
C02384=1084.776,302.489,413.584,176.234,24.553,154.006
C02385=1084.785,302.896,413.533,176.238,24.559,154.007
C02386=1084.794,303.303,413.482,176.244,24.566,154.008
C02387=1084.803,303.710,413.431,176.248,24.572,154.009
C02388=1084.814,304.116,413.380,176.253,24.578,154.010
C02389=1084.819,304.364,413.349,176.256,24.582,154.010
C02390=1084.825,304.611,413.318,176.259,24.586,154.011
C02391=1084.830,304.859,413.287,176.262,24.589,154.011
C02392=1084.836,305.108,413.255,176.265,24.593,154.011
C02393=1084.842,305.355,413.224,176.268,24.597,154.012
C02394=1084.847,305.603,413.193,176.271,24.601,154.012
C02395=1084.854,305.851,413.162,176.274,24.605,154.013
C02396=1084.859,306.099,413.130,176.277,24.608,154.013
C02397=1084.865,306.348,413.099,176.279,24.612,154.014
C02398=1084.871,306.595,413.068,176.282,24.616,154.014
C02399=1084.876,306.843,413.037,176.285,24.620,154.015
C02400=1084.883,307.091,413.005,176.288,24.624,154.015
C02401=1084.888,307.338,412.974,176.291,24.627,154.016
C02402=1084.894,307.587,412.942,176.294,24.631,154.016
C02403=1084.900,307.834,412.911,176.297,24.635,154.017
C02404=1084.906,308.083,412.879,176.300,24.639,154.017
C02405=1084.911,308.331,412.848,176.303,24.642,154.018
C02406=1084.917,308.578,412.817,176.306,24.646,154.018
C02407=1084.923,308.826,412.785,176.309,24.650,154.019
C02408=1084.928,309.074,412.754,176.312,24.654,154.019
C02409=1084.935,309.322,412.723,176.315,24.658,154.020
C02410=1084.940,309.570,412.691,176.317,24.662,154.020
C02411=1084.946,309.818,412.659,176.320,24.665,154.021
C02412=1084.952,310.066,412.629,176.323,24.669,154.021
C02413=1084.958,310.314,412.597,176.326,24.673,154.022
C02414=1084.963,310.561,412.565,176.329,24.677,154.022
C02415=1084.970,310.809,412.534,176.333,24.681,154.023
C02416=1084.976,311.058,412.502,176.336,24.685,154.023
C02417=1084.981,311.305,412.470,176.339,24.689,154.024
C02418=1084.987,311.554,412.439,176.342,24.693,154.024
C02419=1084.993,311.801,412.408,176.345,24.696,154.025
C02420=1084.999,312.049,412.376,176.348,24.700,154.025
C02421=1085.005,312.297,412.344,176.351,24.704,154.026
C02422=1085.011,312.545,412.313,176.354,24.708,154.026
C02423=1085.017,312.793,412.281,176.357,24.712,154.027
C02424=1085.023,313.040,412.249,176.360,24.716,154.027
C02425=1085.029,313.289,412.217,176.363,24.720,154.028
C02426=1085.034,313.536,412.185,176.366,24.723,154.028
C02427=1085.041,313.784,412.154,176.369,24.727,154.029
C02428=1085.047,314.032,412.122,176.372,24.731,154.029
C02429=1085.052,314.280,412.090,176.375,24.735,154.030
C02430=1085.058,314.528,412.058,176.378,24.739,154.030
C02431=1085.065,314.776,412.027,176.380,24.743,154.031
C02432=1085.071,315.024,411.995,176.383,24.747,154.031
C02433=1085.076,315.272,411.962,176.386,24.751,154.032
C02434=1085.082,315.520,411.930,176.389,24.755,154.032
C02435=1085.087,315.767,411.898,176.392,24.759,154.033
C02436=1085.093,316.015,411.866,176.395,24.763,154.033
C02437=1085.102,316.424,411.813,176.400,24.769,154.034
C02438=1085.112,316.835,411.760,176.405,24.776,154.035
C02439=1085.121,317.244,411.707,176.410,24.783,154.036
C02440=1085.130,317.654,411.654,176.415,24.790,154.037
C02441=1085.137,317.901,411.621,176.418,24.794,154.038
C02442=1085.142,318.149,411.590,176.420,24.798,154.038
C02443=1085.147,318.397,411.557,176.423,24.802,154.039
C02444=1085.153,318.645,411.525,176.426,24.806,154.039
C02445=1085.159,318.892,411.493,176.429,24.810,154.040
C02446=1085.165,319.141,411.461,176.432,24.814,154.040
C02447=1085.171,319.389,411.428,176.436,24.818,154.041
C02448=1085.176,319.636,411.396,176.439,24.822,154.042
C02449=1085.182,319.884,411.363,176.442,24.826,154.042
C02450=1085.188,320.132,411.331,176.445,24.830,154.043
C02451=1085.194,320.380,411.299,176.448,24.834,154.043
C02452=1085.199,320.628,411.266,176.450,24.839,154.044
C02453=1085.205,320.875,411.234,176.453,24.843,154.044
C02454=1085.211,321.124,411.202,176.456,24.847,154.045
C02455=1085.216,321.371,411.169,176.459,24.851,154.045
C02456=1085.222,321.619,411.137,176.462,24.855,154.046
C02457=1085.228,321.867,411.104,176.466,24.860,154.047
C02458=1085.234,322.115,411.072,176.469,24.864,154.047
C02459=1085.240,322.363,411.039,176.472,24.868,154.048
C02460=1085.245,322.610,411.006,176.475,24.872,154.048
C02461=1085.251,322.858,410.974,176.477,24.876,154.049
C02462=1085.257,323.106,410.941,176.480,24.880,154.049
C02463=1085.263,323.354,410.909,176.483,24.884,154.050
C02464=1085.269,323.602,410.876,176.486,24.888,154.051
C02465=1085.274,323.849,410.843,176.489,24.892,154.051
C02466=1085.280,324.097,410.811,176.493,24.897,154.052
C02467=1085.287,324.345,410.778,176.496,24.901,154.052
C02468=1085.292,324.592,410.745,176.498,24.905,154.053
C02469=1085.298,324.841,410.713,176.501,24.909,154.054
C02470=1085.304,325.088,410.680,176.504,24.913,154.054
C02471=1085.310,325.336,410.647,176.507,24.918,154.055
C02472=1085.316,325.584,410.614,176.510,24.922,154.055
C02473=1085.321,325.832,410.582,176.514,24.926,154.056
C02474=1085.327,326.079,410.549,176.517,24.930,154.056
C02475=1085.333,326.327,410.516,176.520,24.934,154.057
C02476=1085.339,326.575,410.483,176.523,24.938,154.058
C02477=1085.345,326.822,410.450,176.525,24.943,154.058
C02478=1085.351,327.071,410.418,176.528,24.947,154.059
C02479=1085.357,327.318,410.385,176.532,24.952,154.059
C02480=1085.363,327.566,410.352,176.535,24.956,154.060
C02481=1085.369,327.814,410.319,176.538,24.960,154.061
C02482=1085.375,328.061,410.286,176.541,24.964,154.061
C02483=1085.381,328.309,410.253,176.544,24.968,154.062
C02484=1085.387,328.557,410.220,176.546,24.972,154.062
C02485=1085.392,328.805,410.187,176.550,24.977,154.063
C02486=1085.399,329.052,410.154,176.553,24.981,154.064
C02487=1085.405,329.300,410.121,176.556,24.985,154.064
C02488=1085.411,329.548,410.088,176.559,24.989,154.065
C02489=1085.418,329.854,410.048,176.563,24.994,154.065
C02490=1085.425,330.161,410.007,176.567,25.000,154.066
C02491=1085.432,330.467,409.965,176.571,25.005,154.067
C02492=1085.440,330.773,409.925,176.574,25.011,154.068
C02493=1085.446,331.021,409.891,176.577,25.015,154.068
C02494=1085.452,331.269,409.859,176.580,25.019,154.069
C02495=1085.458,331.516,409.825,176.584,25.024,154.070
C02496=1085.464,331.764,409.792,176.587,25.028,154.070
C02497=1085.470,332.012,409.758,176.590,25.032,154.071
C02498=1085.475,332.260,409.725,176.592,25.036,154.071
C02499=1085.482,332.507,409.692,176.595,25.041,154.072
C02500=1085.488,332.755,409.658,176.599,25.046,154.073
C02501=1085.493,333.002,409.625,176.602,25.050,154.073
C02502=1085.499,333.250,409.592,176.605,25.054,154.074
C02503=1085.504,333.498,409.558,176.608,25.058,154.075
C02504=1085.511,333.745,409.525,176.611,25.063,154.075
C02505=1085.516,333.993,409.491,176.614,25.068,154.076
C02506=1085.523,334.242,409.458,176.617,25.072,154.077
C02507=1085.528,334.489,409.424,176.620,25.077,154.077
C02508=1085.534,334.737,409.390,176.623,25.081,154.078
C02509=1085.540,334.985,409.358,176.626,25.085,154.079
C02510=1085.546,335.232,409.324,176.629,25.090,154.079
C02511=1085.552,335.480,409.290,176.632,25.094,154.080
C02512=1085.558,335.727,409.256,176.636,25.099,154.081
C02513=1085.563,335.975,409.223,176.639,25.104,154.081
C02514=1085.569,336.224,409.189,176.641,25.108,154.082
C02515=1085.576,336.470,409.156,176.644,25.112,154.083
C02516=1085.581,336.718,409.122,176.648,25.117,154.083
C02517=1085.587,336.966,409.088,176.651,25.122,154.084
C02518=1085.593,337.214,409.055,176.654,25.126,154.085
C02519=1085.599,337.461,409.021,176.656,25.130,154.085
C02520=1085.605,337.709,408.987,176.660,25.135,154.086
C02521=1085.614,338.053,408.940,176.665,25.141,154.087
C02522=1085.621,338.397,408.893,176.669,25.148,154.088
C02523=1085.630,338.741,408.846,176.673,25.154,154.089
C02524=1085.638,339.086,408.799,176.677,25.161,154.090
C02525=1085.644,339.333,408.765,176.680,25.165,154.090
C02526=1085.649,339.580,408.731,176.683,25.170,154.091
C02527=1085.656,339.829,408.698,176.686,25.175,154.092
C02528=1085.661,340.076,408.663,176.689,25.179,154.093
C02529=1085.667,340.323,408.629,176.692,25.184,154.093
C02530=1085.672,340.571,408.595,176.695,25.188,154.094
C02531=1085.679,340.820,408.561,176.699,25.194,154.095
C02532=1085.684,341.067,408.527,176.702,25.198,154.095
C02533=1085.690,341.314,408.493,176.704,25.202,154.096
C02534=1085.696,341.561,408.459,176.708,25.207,154.097
C02535=1085.703,341.809,408.425,176.711,25.212,154.097
C02536=1085.708,342.057,408.391,176.714,25.217,154.098
C02537=1085.714,342.305,408.357,176.717,25.221,154.099
C02538=1085.720,342.552,408.323,176.720,25.226,154.100
C02539=1085.726,342.800,408.288,176.723,25.231,154.100
C02540=1085.731,343.047,408.254,176.727,25.235,154.101
C02541=1085.741,343.445,408.199,176.732,25.243,154.102
C02542=1085.751,343.842,408.144,176.737,25.251,154.103
C02543=1085.760,344.239,408.089,176.742,25.258,154.104
C02544=1085.770,344.636,408.034,176.747,25.266,154.106
C02545=1085.776,344.884,408.000,176.750,25.271,154.106
C02546=1085.782,345.131,407.965,176.752,25.276,154.107
C02547=1085.787,345.378,407.931,176.756,25.280,154.108
C02548=1085.794,345.626,407.896,176.759,25.285,154.109
C02549=1085.800,345.873,407.862,176.762,25.291,154.109
C02550=1085.805,346.121,407.827,176.765,25.295,154.110
C02551=1085.811,346.369,407.793,176.768,25.300,154.111
C02552=1085.817,346.616,407.759,176.772,25.305,154.112
C02553=1085.823,346.863,407.724,176.774,25.310,154.112
C02554=1085.829,347.111,407.689,176.777,25.314,154.113
C02555=1085.835,347.359,407.655,176.781,25.320,154.114
C02556=1085.841,347.607,407.620,176.784,25.324,154.115
C02557=1085.847,347.854,407.585,176.787,25.329,154.115
C02558=1085.853,348.101,407.551,176.790,25.334,154.116
C02559=1085.858,348.349,407.516,176.793,25.339,154.117
C02560=1085.864,348.596,407.482,176.796,25.344,154.118
C02561=1085.870,348.844,407.447,176.799,25.349,154.119
C02562=1085.876,349.091,407.412,176.803,25.354,154.119
C02563=1085.882,349.339,407.377,176.805,25.359,154.120
C02564=1085.888,349.586,407.343,176.809,25.364,154.121
C02565=1085.894,349.835,407.308,176.812,25.369,154.122
C02566=1085.900,350.081,407.273,176.815,25.374,154.123
C02567=1085.906,350.329,407.239,176.818,25.379,154.123
C02568=1085.912,350.576,407.203,176.821,25.384,154.124
C02569=1085.918,350.824,407.169,176.825,25.389,154.125
C02570=1085.924,351.071,407.133,176.827,25.394,154.126
C02571=1085.930,351.319,407.099,176.831,25.399,154.126
C02572=1085.936,351.566,407.064,176.834,25.404,154.127
C02573=1085.942,351.814,407.029,176.837,25.409,154.128
C02574=1085.947,352.061,406.994,176.840,25.414,154.129
C02575=1085.953,352.309,406.959,176.843,25.419,154.130
C02576=1085.959,352.556,406.924,176.846,25.425,154.130
C02577=1085.965,352.804,406.888,176.849,25.429,154.131
C02578=1085.971,353.051,406.854,176.853,25.435,154.132
C02579=1085.977,353.299,406.818,176.856,25.440,154.133
C02580=1085.983,353.546,406.783,176.859,25.445,154.134
C02581=1085.989,353.794,406.749,176.862,25.450,154.134
C02582=1085.995,354.041,406.713,176.866,25.455,154.135
C02583=1086.001,354.288,406.678,176.868,25.460,154.136
C02584=1086.007,354.536,406.642,176.872,25.465,154.137
C02585=1086.012,354.783,406.608,176.875,25.471,154.138
C02586=1086.019,355.031,406.572,176.878,25.476,154.139
C02587=1086.025,355.278,406.537,176.881,25.481,154.140
C02588=1086.031,355.525,406.502,176.884,25.487,154.140
C02589=1086.037,355.773,406.466,176.887,25.492,154.141
C02590=1086.042,356.021,406.431,176.891,25.497,154.142
C02591=1086.049,356.268,406.396,176.893,25.502,154.143
C02592=1086.055,356.516,406.360,176.897,25.507,154.144
C02593=1086.064,356.915,406.303,176.902,25.516,154.145
C02594=1086.074,357.315,406.246,176.907,25.525,154.147
C02595=1086.083,357.715,406.188,176.912,25.533,154.148
C02596=1086.093,358.115,406.131,176.917,25.542,154.149
C02597=1086.099,358.362,406.096,176.920,25.547,154.150
C02598=1086.105,358.610,406.060,176.924,25.552,154.151
C02599=1086.112,358.857,406.024,176.927,25.558,154.152
C02600=1086.117,359.104,405.989,176.930,25.563,154.153
C02601=1086.123,359.352,405.953,176.933,25.569,154.154
C02602=1086.129,359.599,405.917,176.936,25.574,154.155
C02603=1086.135,359.847,405.882,176.940,25.579,154.156
C02604=1086.141,360.094,405.846,176.942,25.584,154.156
C02605=1086.147,360.342,405.810,176.946,25.590,154.157
C02606=1086.153,360.589,405.774,176.949,25.595,154.158
C02607=1086.159,360.836,405.739,176.952,25.601,154.159
C02608=1086.165,361.083,405.704,176.956,25.606,154.160
C02609=1086.171,361.331,405.668,176.958,25.612,154.161
C02610=1086.178,361.578,405.631,176.962,25.617,154.162
C02611=1086.184,361.825,405.596,176.965,25.623,154.163
C02612=1086.189,362.072,405.560,176.968,25.628,154.164
C02613=1086.196,362.319,405.524,176.971,25.634,154.165
C02614=1086.202,362.567,405.488,176.974,25.639,154.166
C02615=1086.208,362.815,405.452,176.978,25.645,154.167
C02616=1086.214,363.062,405.416,176.981,25.650,154.168
C02617=1086.219,363.309,405.381,176.984,25.656,154.168
C02618=1086.225,363.556,405.345,176.987,25.661,154.169
C02619=1086.231,363.804,405.308,176.990,25.667,154.170
C02620=1086.237,364.051,405.272,176.994,25.673,154.171
C02621=1086.243,364.299,405.236,176.997,25.678,154.172
C02622=1086.249,364.546,405.200,177.000,25.684,154.173
C02623=1086.255,364.793,405.164,177.003,25.690,154.174
C02624=1086.261,365.040,405.128,177.006,25.695,154.175
C02625=1086.267,365.287,405.092,177.010,25.701,154.176
C02626=1086.274,365.534,405.055,177.012,25.706,154.177
C02627=1086.280,365.782,405.019,177.016,25.712,154.178
C02628=1086.285,366.029,404.982,177.019,25.718,154.179
C02629=1086.291,366.277,404.947,177.022,25.724,154.180
C02630=1086.297,366.523,404.911,177.026,25.730,154.181
C02631=1086.304,366.770,404.874,177.028,25.735,154.182
C02632=1086.309,367.018,404.837,177.032,25.741,154.183
C02633=1086.315,367.265,404.801,177.035,25.747,154.184
C02634=1086.322,367.513,404.765,177.038,25.752,154.185
C02635=1086.327,367.760,404.728,177.041,25.759,154.186
C02636=1086.333,368.007,404.691,177.045,25.764,154.187
C02637=1086.339,368.255,404.656,177.047,25.770,154.188
C02638=1086.345,368.502,404.619,177.051,25.776,154.189
C02639=1086.351,368.749,404.582,177.054,25.782,154.190
C02640=1086.358,368.996,404.546,177.057,25.788,154.191
C02641=1086.363,369.243,404.509,177.061,25.793,154.192
C02642=1086.369,369.490,404.473,177.064,25.799,154.193
C02643=1086.375,369.737,404.436,177.067,25.805,154.194
C02644=1086.381,369.985,404.400,177.070,25.811,154.195
C02645=1086.392,370.400,404.338,177.076,25.821,154.197
C02646=1086.402,370.816,404.277,177.081,25.831,154.198
C02647=1086.412,371.232,404.214,177.087,25.841,154.200
C02648=1086.422,371.648,404.153,177.092,25.851,154.202
C02649=1086.429,371.895,404.117,177.095,25.857,154.203
C02650=1086.435,372.141,404.079,177.098,25.863,154.204
C02651=1086.441,372.389,404.042,177.102,25.869,154.205
C02652=1086.447,372.636,404.005,177.105,25.875,154.206
C02653=1086.453,372.883,403.969,177.108,25.881,154.207
C02654=1086.459,373.130,403.932,177.111,25.887,154.208
C02655=1086.465,373.377,403.895,177.115,25.893,154.209
C02656=1086.472,373.624,403.858,177.118,25.900,154.210
C02657=1086.477,373.871,403.821,177.121,25.905,154.211
C02658=1086.483,374.118,403.785,177.124,25.911,154.212
C02659=1086.489,374.366,403.748,177.127,25.918,154.214
C02660=1086.496,374.613,403.710,177.131,25.924,154.215
C02661=1086.502,374.860,403.673,177.133,25.930,154.216
C02662=1086.507,375.107,403.636,177.137,25.937,154.217
C02663=1086.513,375.354,403.598,177.140,25.943,154.218
C02664=1086.520,375.601,403.562,177.144,25.949,154.219
C02665=1086.525,375.849,403.525,177.146,25.955,154.220
C02666=1086.531,376.095,403.487,177.150,25.962,154.221
C02667=1086.538,376.342,403.451,177.153,25.968,154.223
C02668=1086.543,376.589,403.413,177.157,25.974,154.224
C02669=1086.550,376.837,403.376,177.159,25.981,154.225
C02670=1086.556,377.084,403.338,177.163,25.987,154.226
C02671=1086.562,377.331,403.301,177.166,25.993,154.227
C02672=1086.568,377.578,403.264,177.169,26.000,154.228
C02673=1086.573,377.825,403.227,177.173,26.006,154.229
C02674=1086.580,378.072,403.189,177.175,26.012,154.231
C02675=1086.587,378.319,403.151,177.179,26.019,154.232
C02676=1086.592,378.566,403.114,177.182,26.025,154.233
C02677=1086.598,378.813,403.077,177.186,26.031,154.234
C02678=1086.604,379.060,403.040,177.189,26.038,154.235
C02679=1086.610,379.307,403.002,177.192,26.045,154.236
C02680=1086.617,379.554,402.964,177.195,26.051,154.238
C02681=1086.623,379.801,402.926,177.198,26.057,154.239
C02682=1086.629,380.048,402.890,177.202,26.064,154.240
C02683=1086.636,380.296,402.852,177.205,26.071,154.241
C02684=1086.641,380.542,402.814,177.208,26.077,154.242
C02685=1086.647,380.789,402.776,177.212,26.084,154.243
C02686=1086.653,381.036,402.739,177.214,26.090,154.245
C02687=1086.660,381.284,402.702,177.218,26.096,154.246
C02688=1086.666,381.530,402.664,177.221,26.103,154.247
C02689=1086.672,381.777,402.626,177.225,26.110,154.248
C02690=1086.679,382.025,402.588,177.228,26.116,154.249
C02691=1086.684,382.271,402.550,177.231,26.123,154.251
C02692=1086.691,382.519,402.512,177.235,26.130,154.252
C02693=1086.697,382.765,402.475,177.238,26.136,154.253
C02694=1086.703,383.012,402.437,177.241,26.143,154.254
C02695=1086.709,383.259,402.399,177.244,26.150,154.256
C02696=1086.715,383.506,402.361,177.247,26.156,154.257
C02697=1086.720,383.728,402.327,177.251,26.163,154.258
C02698=1086.726,383.949,402.293,177.253,26.168,154.259
C02699=1086.731,384.171,402.259,177.257,26.175,154.260
C02700=1086.737,384.393,402.224,177.259,26.181,154.261
C02701=1086.742,384.615,402.191,177.262,26.187,154.262
C02702=1086.748,384.838,402.156,177.265,26.193,154.264
C02703=1086.753,385.059,402.123,177.268,26.199,154.265
C02704=1086.759,385.281,402.088,177.271,26.206,154.266
C02705=1086.765,385.527,402.050,177.275,26.213,154.267
C02706=1086.772,385.774,402.012,177.277,26.219,154.268
C02707=1086.777,386.021,401.973,177.280,26.226,154.270
C02708=1086.783,386.269,401.935,177.284,26.233,154.271
C02709=1086.789,386.515,401.897,177.287,26.240,154.272
C02710=1086.795,386.762,401.859,177.290,26.247,154.274
C02711=1086.802,387.009,401.821,177.294,26.254,154.275
C02712=1086.808,387.255,401.783,177.297,26.261,154.276
C02713=1086.815,387.503,401.744,177.300,26.268,154.278
C02714=1086.821,387.749,401.707,177.304,26.275,154.279
C02715=1086.827,387.997,401.667,177.307,26.282,154.280
C02716=1086.832,388.243,401.629,177.310,26.289,154.281
C02717=1086.839,388.490,401.591,177.314,26.296,154.283
C02718=1086.845,388.737,401.553,177.317,26.303,154.284
C02719=1086.852,388.984,401.514,177.320,26.310,154.286
C02720=1086.857,389.231,401.476,177.324,26.317,154.287
C02721=1086.864,389.478,401.437,177.327,26.324,154.288
C02722=1086.870,389.724,401.399,177.330,26.331,154.289
C02723=1086.877,389.971,401.360,177.333,26.339,154.291
C02724=1086.883,390.219,401.322,177.337,26.346,154.292
C02725=1086.889,390.465,401.283,177.340,26.353,154.294
C02726=1086.896,390.712,401.244,177.343,26.360,154.295
C02727=1086.901,390.959,401.206,177.347,26.367,154.296
C02728=1086.908,391.205,401.168,177.350,26.375,154.298
C02729=1086.914,391.453,401.128,177.353,26.382,154.299
C02730=1086.920,391.699,401.090,177.357,26.389,154.300
C02731=1086.927,391.946,401.052,177.361,26.397,154.302
C02732=1086.933,392.193,401.012,177.364,26.404,154.303
C02733=1086.939,392.439,400.974,177.367,26.412,154.305
C02734=1086.945,392.686,400.934,177.371,26.419,154.306
C02735=1086.952,392.934,400.896,177.374,26.426,154.308
C02736=1086.957,393.180,400.857,177.377,26.434,154.309
C02737=1086.964,393.427,400.818,177.380,26.441,154.310
C02738=1086.971,393.674,400.779,177.384,26.449,154.312
C02739=1086.976,393.920,400.740,177.387,26.456,154.313
C02740=1086.983,394.167,400.702,177.390,26.464,154.315
C02741=1086.989,394.414,400.662,177.393,26.471,154.316
C02742=1086.996,394.661,400.624,177.397,26.479,154.318
C02743=1087.002,394.908,400.584,177.400,26.486,154.319
C02744=1087.008,395.155,400.545,177.404,26.494,154.321
C02745=1087.014,395.402,400.506,177.407,26.502,154.322
C02746=1087.020,395.648,400.467,177.411,26.509,154.323
C02747=1087.027,395.895,400.428,177.414,26.517,154.325
C02748=1087.033,396.142,400.389,177.417,26.525,154.326
C02749=1087.039,396.389,400.349,177.420,26.533,154.328
C02750=1087.045,396.635,400.311,177.423,26.540,154.329
C02751=1087.051,396.882,400.271,177.427,26.548,154.331
C02752=1087.058,397.129,400.231,177.430,26.555,154.332
C02753=1087.064,397.358,400.195,177.433,26.563,154.334
C02754=1087.069,397.587,400.159,177.437,26.570,154.335
C02755=1087.076,397.815,400.122,177.440,26.578,154.337
C02756=1087.081,398.044,400.086,177.443,26.585,154.338
C02757=1087.087,398.272,400.049,177.446,26.592,154.340
C02758=1087.093,398.501,400.013,177.449,26.599,154.341
C02759=1087.098,398.729,399.976,177.452,26.606,154.342
C02760=1087.105,398.958,399.940,177.455,26.614,154.344
C02761=1087.111,399.205,399.900,177.459,26.622,154.345
C02762=1087.117,399.452,399.860,177.462,26.630,154.347
C02763=1087.123,399.699,399.821,177.465,26.638,154.349
C02764=1087.130,399.945,399.781,177.469,26.646,154.350
C02765=1087.135,400.192,399.742,177.472,26.654,154.352
C02766=1087.142,400.438,399.702,177.475,26.662,154.353
C02767=1087.148,400.685,399.663,177.479,26.670,154.355
C02768=1087.155,400.932,399.623,177.482,26.678,154.357
C02769=1087.161,401.179,399.583,177.486,26.687,154.358
C02770=1087.167,401.425,399.543,177.489,26.694,154.360
C02771=1087.173,401.673,399.503,177.492,26.703,154.361
C02772=1087.180,401.919,399.463,177.495,26.711,154.363
C02773=1087.186,402.166,399.423,177.499,26.719,154.365
C02774=1087.192,402.413,399.384,177.503,26.728,154.366
C02775=1087.198,402.659,399.344,177.506,26.736,154.368
C02776=1087.205,402.906,399.303,177.509,26.744,154.370
C02777=1087.212,403.153,399.265,177.513,26.753,154.371
C02778=1087.218,403.399,399.224,177.516,26.760,154.373
C02779=1087.224,403.646,399.184,177.519,26.769,154.375
C02780=1087.231,403.892,399.144,177.523,26.777,154.376
C02781=1087.237,404.139,399.105,177.527,26.786,154.378
C02782=1087.244,404.386,399.064,177.530,26.794,154.380
C02783=1087.249,404.633,399.024,177.534,26.803,154.381
C02784=1087.256,404.880,398.983,177.537,26.811,154.383
C02785=1087.262,405.126,398.943,177.540,26.819,154.385
C02786=1087.269,405.373,398.903,177.544,26.828,154.386
C02787=1087.275,405.619,398.863,177.547,26.837,154.388
C02788=1087.281,405.866,398.823,177.550,26.845,154.390
C02789=1087.288,406.112,398.783,177.554,26.854,154.392
C02790=1087.294,406.359,398.742,177.557,26.863,154.393
C02791=1087.300,406.606,398.701,177.561,26.871,154.395
C02792=1087.307,406.853,398.661,177.565,26.880,154.397
C02793=1087.313,407.099,398.621,177.568,26.889,154.399
C02794=1087.319,407.346,398.581,177.572,26.898,154.400
C02795=1087.326,407.592,398.541,177.575,26.906,154.402
C02796=1087.332,407.840,398.500,177.579,26.916,154.404
C02797=1087.338,408.087,398.460,177.582,26.924,154.406
C02798=1087.345,408.332,398.419,177.585,26.933,154.408
C02799=1087.351,408.579,398.378,177.589,26.942,154.409
C02800=1087.357,408.826,398.338,177.592,26.951,154.411
C02801=1087.364,409.073,398.297,177.596,26.960,154.413
C02802=1087.370,409.319,398.256,177.599,26.969,154.415
C02803=1087.376,409.566,398.216,177.603,26.978,154.417
C02804=1087.382,409.813,398.175,177.606,26.987,154.419
C02805=1087.389,410.059,398.134,177.610,26.996,154.420
C02806=1087.396,410.306,398.094,177.613,27.005,154.422
C02807=1087.402,410.552,398.052,177.617,27.014,154.424
C02808=1087.408,410.798,398.012,177.620,27.023,154.426
C02809=1087.414,411.028,397.974,177.623,27.032,154.428
C02810=1087.420,411.257,397.936,177.627,27.040,154.430
C02811=1087.427,411.487,397.897,177.631,27.049,154.431
C02812=1087.432,411.716,397.859,177.634,27.057,154.433
C02813=1087.438,411.945,397.822,177.637,27.066,154.435
C02814=1087.444,412.175,397.783,177.640,27.075,154.437
C02815=1087.451,412.404,397.746,177.643,27.083,154.438
C02816=1087.456,412.632,397.707,177.646,27.092,154.440
C02817=1087.462,412.880,397.666,177.650,27.101,154.442
C02818=1087.469,413.126,397.625,177.654,27.111,154.444
C02819=1087.476,413.373,397.583,177.657,27.120,154.446
C02820=1087.482,413.619,397.542,177.661,27.130,154.448
C02821=1087.488,413.866,397.502,177.664,27.139,154.450
C02822=1087.495,414.112,397.460,177.668,27.149,154.452
C02823=1087.501,414.358,397.419,177.672,27.158,154.454
C02824=1087.508,414.605,397.378,177.675,27.167,154.456
C02825=1087.514,414.851,397.336,177.679,27.177,154.458
C02826=1087.521,415.098,397.296,177.683,27.187,154.460
C02827=1087.527,415.345,397.254,177.686,27.196,154.462
C02828=1087.535,415.591,397.213,177.690,27.206,154.464
C02829=1087.541,415.837,397.172,177.694,27.216,154.466
C02830=1087.548,416.084,397.130,177.697,27.225,154.468
C02831=1087.554,416.331,397.089,177.701,27.235,154.470
C02832=1087.560,416.577,397.047,177.705,27.245,154.472
C02833=1087.567,416.824,397.005,177.708,27.255,154.474
C02834=1087.574,417.070,396.964,177.712,27.265,154.476
C02835=1087.580,417.316,396.922,177.716,27.275,154.478
C02836=1087.586,417.562,396.880,177.719,27.284,154.480
C02837=1087.593,417.809,396.839,177.723,27.294,154.482
C02838=1087.599,418.055,396.797,177.727,27.304,154.484
C02839=1087.606,418.302,396.756,177.730,27.314,154.486
C02840=1087.612,418.548,396.714,177.733,27.324,154.489
C02841=1087.619,418.795,396.672,177.737,27.334,154.491
C02842=1087.626,419.041,396.630,177.741,27.345,154.493
C02843=1087.632,419.287,396.588,177.745,27.355,154.495
C02844=1087.638,419.534,396.546,177.749,27.365,154.497
C02845=1087.645,419.780,396.505,177.752,27.375,154.499
C02846=1087.652,420.026,396.463,177.756,27.385,154.501
C02847=1087.658,420.273,396.421,177.760,27.396,154.503
C02848=1087.665,420.519,396.379,177.764,27.406,154.506
C02849=1087.671,420.765,396.337,177.767,27.417,154.508
C02850=1087.678,421.012,396.294,177.771,27.427,154.510
C02851=1087.685,421.259,396.252,177.774,27.437,154.512
C02852=1087.691,421.504,396.210,177.778,27.448,154.514
C02853=1087.697,421.751,396.168,177.782,27.458,154.517
C02854=1087.705,421.997,396.127,177.786,27.468,154.519
C02855=1087.712,422.243,396.084,177.790,27.479,154.521
C02856=1087.718,422.490,396.043,177.794,27.490,154.523
C02857=1087.724,422.736,395.999,177.797,27.500,154.526
C02858=1087.731,422.983,395.957,177.801,27.511,154.528
C02859=1087.738,423.229,395.914,177.805,27.522,154.530
C02860=1087.744,423.475,395.873,177.808,27.532,154.532
C02861=1087.750,423.721,395.830,177.812,27.543,154.535
C02862=1087.757,423.968,395.788,177.816,27.554,154.537
C02863=1087.764,424.214,395.745,177.820,27.564,154.539
C02864=1087.770,424.459,395.703,177.823,27.576,154.542
C02865=1087.777,424.697,395.662,177.827,27.586,154.544
C02866=1087.783,424.933,395.621,177.831,27.596,154.546
C02867=1087.789,425.171,395.580,177.835,27.607,154.548
C02868=1087.796,425.408,395.539,177.838,27.618,154.551
C02869=1087.802,425.645,395.498,177.842,27.628,154.553
C02870=1087.809,425.882,395.457,177.846,27.639,154.555
C02871=1087.815,426.119,395.416,177.850,27.650,154.558
C02872=1087.821,426.356,395.374,177.853,27.660,154.560
C02873=1087.828,426.602,395.331,177.857,27.672,154.562
C02874=1087.835,426.849,395.289,177.861,27.683,154.565
C02875=1087.842,427.095,395.246,177.865,27.694,154.567
C02876=1087.849,427.341,395.204,177.869,27.705,154.570
C02877=1087.855,427.587,395.160,177.873,27.717,154.572
C02878=1087.862,427.833,395.117,177.876,27.728,154.574
C02879=1087.869,428.080,395.075,177.880,27.739,154.577
C02880=1087.876,428.325,395.032,177.884,27.751,154.579
C02881=1087.882,428.572,394.989,177.888,27.762,154.582
C02882=1087.889,428.818,394.946,177.892,27.774,154.584
C02883=1087.895,429.064,394.902,177.895,27.785,154.587
C02884=1087.902,429.310,394.860,177.899,27.797,154.589
C02885=1087.909,429.556,394.816,177.904,27.808,154.592
C02886=1087.916,429.803,394.773,177.908,27.820,154.594
C02887=1087.923,430.048,394.730,177.911,27.832,154.597
C02888=1087.929,430.294,394.686,177.915,27.843,154.599
C02889=1087.936,430.541,394.644,177.919,27.855,154.602
C02890=1087.942,430.787,394.600,177.923,27.867,154.605
C02891=1087.950,431.032,394.556,177.928,27.879,154.607
C02892=1087.956,431.279,394.513,177.931,27.891,154.610
C02893=1087.963,431.525,394.470,177.935,27.903,154.612
C02894=1087.969,431.771,394.426,177.939,27.914,154.615
C02895=1087.976,432.016,394.383,177.943,27.927,154.618
C02896=1087.983,432.263,394.340,177.947,27.939,154.620
C02897=1087.990,432.509,394.296,177.951,27.951,154.623
C02898=1087.997,432.755,394.252,177.955,27.963,154.626
C02899=1088.003,433.001,394.209,177.960,27.975,154.628
C02900=1088.010,433.247,394.165,177.963,27.987,154.631
C02901=1088.017,433.493,394.121,177.967,28.000,154.634
C02902=1088.023,433.739,394.078,177.971,28.012,154.636
C02903=1088.030,433.985,394.033,177.975,28.024,154.639
C02904=1088.037,434.231,393.990,177.979,28.037,154.642
C02905=1088.044,434.477,393.946,177.983,28.049,154.645
C02906=1088.051,434.722,393.902,177.988,28.062,154.647
C02907=1088.057,434.968,393.858,177.991,28.074,154.650
C02908=1088.065,435.215,393.814,177.995,28.087,154.653
C02909=1088.071,435.461,393.770,178.000,28.100,154.656
C02910=1088.078,435.706,393.726,178.003,28.112,154.659
C02911=1088.084,435.952,393.682,178.007,28.125,154.661
C02912=1088.091,436.199,393.638,178.012,28.138,154.664
C02913=1088.099,436.444,393.594,178.016,28.150,154.667
C02914=1088.105,436.690,393.550,178.020,28.163,154.670
C02915=1088.112,436.936,393.506,178.024,28.176,154.673
C02916=1088.119,437.182,393.461,178.028,28.189,154.676
C02917=1088.125,437.428,393.417,178.032,28.202,154.678
C02918=1088.133,437.674,393.372,178.036,28.215,154.681
C02919=1088.140,437.919,393.329,178.041,28.228,154.684
C02920=1088.147,438.165,393.284,178.044,28.241,154.687
C02921=1088.154,438.435,393.235,178.049,28.255,154.690
C02922=1088.162,438.704,393.187,178.053,28.270,154.694
C02923=1088.170,438.973,393.138,178.058,28.284,154.697
C02924=1088.178,439.242,393.090,178.063,28.299,154.700
C02925=1088.185,439.487,393.045,178.067,28.312,154.703
C02926=1088.192,439.734,393.001,178.072,28.326,154.706
C02927=1088.198,439.979,392.956,178.075,28.339,154.709
C02928=1088.206,440.226,392.911,178.080,28.352,154.712
C02929=1088.212,440.471,392.867,178.084,28.366,154.715
C02930=1088.219,440.717,392.821,178.088,28.380,154.718
C02931=1088.226,440.963,392.777,178.092,28.393,154.721
C02932=1088.233,441.209,392.732,178.097,28.407,154.724
C02933=1088.240,441.454,392.687,178.100,28.420,154.728
C02934=1088.247,441.700,392.642,178.105,28.435,154.731
C02935=1088.254,441.945,392.598,178.110,28.448,154.734
C02936=1088.261,442.191,392.553,178.113,28.462,154.737
C02937=1088.269,442.438,392.508,178.118,28.476,154.740
C02938=1088.275,442.683,392.463,178.123,28.490,154.743
C02939=1088.282,442.929,392.417,178.126,28.504,154.746
C02940=1088.289,443.174,392.372,178.131,28.518,154.750
C02941=1088.296,443.420,392.328,178.136,28.532,154.753
C02942=1088.303,443.666,392.281,178.139,28.547,154.756
C02943=1088.310,443.911,392.237,178.144,28.561,154.759
C02944=1088.317,444.157,392.192,178.148,28.576,154.763
C02945=1088.324,444.403,392.146,178.152,28.590,154.766
C02946=1088.331,444.648,392.101,178.157,28.604,154.769
C02947=1088.338,444.894,392.055,178.161,28.619,154.772
C02948=1088.346,445.140,392.010,178.165,28.633,154.776
C02949=1088.353,445.385,391.964,178.169,28.647,154.779
C02950=1088.359,445.631,391.920,178.172,28.662,154.782
C02951=1088.366,445.877,391.873,178.176,28.676,154.786
C02952=1088.374,446.122,391.828,178.179,28.691,154.789
C02953=1088.381,446.368,391.782,178.183,28.705,154.793
C02954=1088.388,446.613,391.737,178.185,28.719,154.796
C02955=1088.395,446.859,391.691,178.187,28.733,154.799
C02956=1088.402,447.104,391.645,178.190,28.748,154.803
C02957=1088.409,447.350,391.600,178.192,28.762,154.806
C02958=1088.416,447.596,391.554,178.194,28.776,154.810
C02959=1088.424,447.842,391.508,178.196,28.791,154.813
C02960=1088.431,448.087,391.462,178.198,28.805,154.817
C02961=1088.438,448.332,391.417,178.199,28.820,154.820
C02962=1088.445,448.578,391.370,178.200,28.833,154.824
C02963=1088.451,448.824,391.325,178.202,28.848,154.827
C02964=1088.459,449.070,391.279,178.203,28.862,154.831
C02965=1088.467,449.314,391.233,178.204,28.876,154.834
C02966=1088.473,449.559,391.187,178.205,28.890,154.838
C02967=1088.482,449.805,391.142,178.206,28.904,154.841
C02968=1088.492,450.051,391.097,178.207,28.917,154.845
C02969=1088.113,450.043,390.903,178.167,29.108,154.897
C02970=1088.103,449.798,390.947,178.165,29.096,154.894
C02971=1088.095,449.552,390.993,178.164,29.082,154.890
C02972=1088.088,449.307,391.038,178.163,29.067,154.887
C02973=1088.080,449.062,391.085,178.162,29.054,154.883
C02974=1088.073,448.817,391.131,178.162,29.039,154.879
C02975=1088.065,448.571,391.176,178.160,29.025,154.876
C02976=1088.058,448.325,391.223,178.159,29.010,154.872
C02977=1088.051,448.080,391.268,178.157,28.996,154.869
C02978=1088.044,447.834,391.314,178.155,28.982,154.865
C02979=1088.036,447.588,391.360,178.153,28.968,154.862
C02980=1088.029,447.342,391.406,178.151,28.954,154.858
C02981=1088.022,447.097,391.451,178.148,28.939,154.855
C02982=1088.016,446.852,391.497,178.146,28.925,154.852
C02983=1088.008,446.607,391.543,178.144,28.910,154.848
C02984=1088.001,446.361,391.589,178.140,28.896,154.845
C02985=1087.994,446.115,391.634,178.137,28.881,154.841
C02986=1087.987,445.869,391.680,178.134,28.867,154.838
C02987=1087.979,445.624,391.726,178.130,28.853,154.835
C02988=1087.973,445.378,391.771,178.127,28.838,154.831
C02989=1087.965,445.133,391.817,178.123,28.824,154.828
C02990=1087.958,444.887,391.862,178.118,28.809,154.824
C02991=1087.951,444.641,391.908,178.114,28.795,154.821
C02992=1087.944,444.395,391.954,178.110,28.780,154.818
C02993=1087.937,444.150,391.998,178.105,28.766,154.815
C02994=1087.930,443.904,392.044,178.101,28.751,154.811
C02995=1087.923,443.658,392.089,178.096,28.737,154.808
C02996=1087.916,443.413,392.135,178.092,28.723,154.805
C02997=1087.908,443.167,392.180,178.088,28.709,154.802
C02998=1087.902,442.921,392.225,178.083,28.695,154.798
C02999=1087.895,442.676,392.270,178.078,28.680,154.795
C03000=1087.887,442.430,392.315,178.075,28.667,154.792
C03001=1087.881,442.185,392.360,178.070,28.652,154.789
C03002=1087.874,441.939,392.405,178.065,28.638,154.786
C03003=1087.866,441.693,392.451,178.061,28.625,154.783
C03004=1087.860,441.448,392.496,178.057,28.611,154.779
C03005=1087.852,441.202,392.541,178.053,28.597,154.776
C03006=1087.846,440.956,392.585,178.048,28.583,154.773
C03007=1087.838,440.710,392.630,178.044,28.570,154.770
C03008=1087.831,440.464,392.675,178.040,28.556,154.767
C03009=1087.824,440.219,392.720,178.035,28.542,154.764
C03010=1087.817,439.973,392.764,178.031,28.529,154.761
C03011=1087.810,439.727,392.809,178.026,28.515,154.758
C03012=1087.803,439.481,392.854,178.023,28.502,154.755
C03013=1087.796,439.235,392.898,178.018,28.488,154.752
C03014=1087.789,438.979,392.945,178.014,28.475,154.749
C03015=1087.781,438.723,392.991,178.009,28.461,154.746
C03016=1087.774,438.468,393.037,178.005,28.447,154.743
C03017=1087.767,438.211,393.083,178.000,28.433,154.740
C03018=1087.760,437.966,393.128,177.996,28.421,154.737
C03019=1087.753,437.719,393.173,177.992,28.408,154.734
C03020=1087.746,437.474,393.217,177.988,28.394,154.731
C03021=1087.740,437.228,393.261,177.984,28.381,154.728
C03022=1087.732,436.981,393.306,177.979,28.368,154.725
C03023=1087.726,436.736,393.350,177.975,28.355,154.722
C03024=1087.719,436.490,393.393,177.971,28.343,154.719
C03025=1087.711,436.244,393.438,177.967,28.330,154.716
C03026=1087.705,435.998,393.482,177.963,28.317,154.714
C03027=1087.698,435.753,393.527,177.958,28.304,154.711
C03028=1087.691,435.506,393.571,177.954,28.291,154.708
C03029=1087.684,435.261,393.614,177.951,28.279,154.705
C03030=1087.678,435.015,393.658,177.946,28.266,154.702
C03031=1087.670,434.769,393.703,177.942,28.254,154.700
C03032=1087.664,434.523,393.747,177.938,28.241,154.697
C03033=1087.657,434.277,393.791,177.933,28.228,154.694
C03034=1087.650,434.031,393.834,177.930,28.216,154.691
C03035=1087.643,433.784,393.878,177.926,28.204,154.688
C03036=1087.636,433.539,393.923,177.922,28.191,154.686
C03037=1087.630,433.293,393.967,177.917,28.179,154.683
C03038=1087.623,433.047,394.010,177.913,28.167,154.680
C03039=1087.616,432.801,394.054,177.909,28.155,154.678
C03040=1087.610,432.556,394.098,177.906,28.143,154.675
C03041=1087.602,432.309,394.141,177.901,28.130,154.672
C03042=1087.596,432.063,394.184,177.897,28.118,154.670
C03043=1087.589,431.817,394.228,177.893,28.106,154.667
C03044=1087.583,431.571,394.271,177.889,28.094,154.664
C03045=1087.575,431.325,394.315,177.884,28.082,154.662
C03046=1087.569,431.079,394.358,177.881,28.070,154.659
C03047=1087.561,430.833,394.402,177.877,28.058,154.657
C03048=1087.555,430.586,394.445,177.873,28.046,154.654
C03049=1087.548,430.341,394.488,177.869,28.035,154.651
C03050=1087.541,430.095,394.532,177.865,28.023,154.649
C03051=1087.535,429.848,394.575,177.860,28.011,154.646
C03052=1087.528,429.602,394.619,177.857,27.999,154.644
C03053=1087.521,429.357,394.662,177.853,27.988,154.641
C03054=1087.515,429.110,394.705,177.849,27.976,154.639
C03055=1087.508,428.865,394.748,177.845,27.965,154.636
C03056=1087.501,428.618,394.791,177.841,27.953,154.634
C03057=1087.494,428.372,394.835,177.837,27.942,154.631
C03058=1087.488,428.126,394.877,177.833,27.930,154.629
C03059=1087.481,427.880,394.920,177.830,27.919,154.626
C03060=1087.474,427.634,394.964,177.826,27.907,154.624
C03061=1087.467,427.387,395.006,177.821,27.896,154.621
C03062=1087.461,427.141,395.049,177.817,27.884,154.619
C03063=1087.453,426.895,395.092,177.813,27.873,154.616
C03064=1087.447,426.649,395.135,177.809,27.862,154.614
C03065=1087.440,426.403,395.178,177.805,27.851,154.612
C03066=1087.434,426.165,395.219,177.801,27.840,154.609
C03067=1087.427,425.928,395.260,177.798,27.830,154.607
C03068=1087.421,425.690,395.301,177.794,27.819,154.605
C03069=1087.415,425.453,395.343,177.790,27.808,154.602
C03070=1087.409,425.215,395.384,177.786,27.797,154.600
C03071=1087.402,424.977,395.424,177.783,27.787,154.598
C03072=1087.395,424.740,395.466,177.779,27.776,154.596
C03073=1087.389,424.502,395.507,177.776,27.766,154.593
C03074=1087.382,424.256,395.550,177.772,27.755,154.591
C03075=1087.375,424.010,395.592,177.768,27.744,154.589
C03076=1087.369,423.763,395.635,177.764,27.733,154.586
C03077=1087.362,423.517,395.677,177.760,27.722,154.584
C03078=1087.356,423.271,395.720,177.756,27.711,154.582
C03079=1087.350,423.024,395.762,177.752,27.701,154.579
C03080=1087.343,422.778,395.804,177.749,27.690,154.577
C03081=1087.336,422.532,395.847,177.745,27.680,154.575
C03082=1087.329,422.286,395.889,177.741,27.669,154.573
C03083=1087.323,422.040,395.932,177.737,27.658,154.570
C03084=1087.316,421.793,395.973,177.733,27.647,154.568
C03085=1087.309,421.547,396.016,177.729,27.637,154.566
C03086=1087.303,421.300,396.058,177.725,27.627,154.564
C03087=1087.297,421.054,396.100,177.722,27.616,154.562
C03088=1087.290,420.808,396.142,177.719,27.606,154.559
C03089=1087.283,420.561,396.184,177.715,27.596,154.557
C03090=1087.276,420.315,396.226,177.711,27.585,154.555
C03091=1087.270,420.069,396.268,177.707,27.575,154.553
C03092=1087.263,419.823,396.310,177.703,27.565,154.551
C03093=1087.256,419.576,396.352,177.700,27.554,154.548
C03094=1087.250,419.330,396.394,177.696,27.544,154.546
C03095=1087.244,419.083,396.436,177.692,27.534,154.544
C03096=1087.237,418.836,396.478,177.688,27.524,154.542
C03097=1087.230,418.591,396.519,177.685,27.514,154.540
C03098=1087.223,418.344,396.561,177.681,27.504,154.538
C03099=1087.217,418.098,396.603,177.677,27.494,154.536
C03100=1087.211,417.852,396.645,177.673,27.483,154.533
C03101=1087.204,417.605,396.687,177.670,27.474,154.531
C03102=1087.198,417.359,396.729,177.666,27.464,154.529
C03103=1087.191,417.112,396.770,177.662,27.454,154.527
C03104=1087.185,416.866,396.811,177.658,27.444,154.525
C03105=1087.178,416.619,396.854,177.655,27.434,154.523
C03106=1087.172,416.373,396.895,177.651,27.424,154.521
C03107=1087.165,416.127,396.936,177.647,27.414,154.519
C03108=1087.159,415.880,396.978,177.644,27.404,154.517
C03109=1087.152,415.634,397.020,177.640,27.394,154.515
C03110=1087.145,415.387,397.061,177.636,27.385,154.513
C03111=1087.139,415.141,397.102,177.633,27.375,154.511
C03112=1087.132,414.894,397.144,177.629,27.366,154.509
C03113=1087.126,414.648,397.185,177.625,27.356,154.507
C03114=1087.119,414.401,397.226,177.622,27.347,154.505
C03115=1087.113,414.155,397.267,177.618,27.337,154.503
C03116=1087.106,413.908,397.308,177.615,27.327,154.501
C03117=1087.100,413.662,397.350,177.611,27.318,154.499
C03118=1087.092,413.415,397.391,177.607,27.308,154.497
C03119=1087.087,413.168,397.432,177.604,27.299,154.495
C03120=1087.080,412.922,397.473,177.600,27.290,154.493
C03121=1087.073,412.676,397.514,177.596,27.280,154.491
C03122=1087.068,412.446,397.553,177.593,27.272,154.489
C03123=1087.062,412.216,397.591,177.589,27.263,154.488
C03124=1087.055,411.986,397.629,177.586,27.254,154.486
C03125=1087.049,411.756,397.667,177.583,27.246,154.484
C03126=1087.043,411.527,397.705,177.580,27.237,154.482
C03127=1087.037,411.297,397.744,177.576,27.229,154.481
C03128=1087.032,411.067,397.782,177.573,27.220,154.479
C03129=1087.025,410.837,397.821,177.569,27.211,154.477
C03130=1087.019,410.590,397.861,177.566,27.202,154.475
C03131=1087.012,410.344,397.902,177.562,27.193,154.473
C03132=1087.006,410.097,397.943,177.559,27.184,154.471
C03133=1086.999,409.851,397.984,177.556,27.175,154.470
C03134=1086.994,409.604,398.024,177.552,27.165,154.468
C03135=1086.987,409.358,398.064,177.548,27.157,154.466
C03136=1086.980,409.111,398.106,177.544,27.148,154.464
C03137=1086.974,408.864,398.146,177.541,27.139,154.462
C03138=1086.968,408.618,398.187,177.537,27.129,154.460
C03139=1086.962,408.371,398.228,177.534,27.120,154.458
C03140=1086.955,408.124,398.269,177.530,27.111,154.457
C03141=1086.949,407.878,398.309,177.527,27.103,154.455
C03142=1086.943,407.631,398.349,177.524,27.094,154.453
C03143=1086.936,407.385,398.390,177.520,27.085,154.451
C03144=1086.930,407.138,398.430,177.516,27.076,154.450
C03145=1086.923,406.891,398.471,177.512,27.067,154.448
C03146=1086.916,406.645,398.511,177.509,27.059,154.446
C03147=1086.911,406.398,398.552,177.506,27.050,154.444
C03148=1086.904,406.151,398.592,177.502,27.041,154.442
C03149=1086.898,405.905,398.632,177.499,27.033,154.441
C03150=1086.892,405.658,398.672,177.496,27.024,154.439
C03151=1086.885,405.411,398.713,177.492,27.015,154.437
C03152=1086.878,405.165,398.753,177.488,27.007,154.436
C03153=1086.873,404.918,398.794,177.485,26.998,154.434
C03154=1086.866,404.671,398.834,177.481,26.990,154.432
C03155=1086.860,404.425,398.874,177.478,26.981,154.430
C03156=1086.854,404.178,398.914,177.475,26.973,154.429
C03157=1086.847,403.932,398.954,177.471,26.964,154.427
C03158=1086.841,403.685,398.994,177.467,26.956,154.425
C03159=1086.835,403.438,399.034,177.464,26.948,154.424
C03160=1086.828,403.191,399.074,177.460,26.939,154.422
C03161=1086.821,402.944,399.115,177.457,26.931,154.420
C03162=1086.815,402.698,399.155,177.454,26.922,154.419
C03163=1086.809,402.451,399.194,177.451,26.914,154.417
C03164=1086.803,402.204,399.234,177.446,26.906,154.415
C03165=1086.795,401.958,399.274,177.443,26.897,154.414
C03166=1086.789,401.711,399.313,177.440,26.890,154.412
C03167=1086.783,401.464,399.353,177.437,26.881,154.410
C03168=1086.777,401.218,399.394,177.433,26.873,154.409
C03169=1086.770,400.971,399.433,177.429,26.865,154.407
C03170=1086.764,400.724,399.473,177.426,26.857,154.406
C03171=1086.758,400.477,399.513,177.423,26.849,154.404
C03172=1086.752,400.230,399.553,177.420,26.841,154.402
C03173=1086.746,399.983,399.592,177.416,26.832,154.401
C03174=1086.740,399.738,399.632,177.412,26.824,154.399
C03175=1086.733,399.491,399.671,177.409,26.816,154.398
C03176=1086.727,399.244,399.711,177.406,26.808,154.396
C03177=1086.721,398.997,399.750,177.403,26.800,154.394
C03178=1086.715,398.768,399.787,177.399,26.793,154.393
C03179=1086.709,398.538,399.823,177.396,26.786,154.392
C03180=1086.703,398.310,399.860,177.393,26.778,154.390
C03181=1086.696,398.080,399.897,177.389,26.771,154.389
C03182=1086.691,397.851,399.934,177.387,26.764,154.387
C03183=1086.685,397.621,399.970,177.384,26.756,154.386
C03184=1086.679,397.393,400.008,177.380,26.749,154.384
C03185=1086.673,397.164,400.044,177.377,26.741,154.383
C03186=1086.667,396.917,400.083,177.374,26.734,154.381
C03187=1086.661,396.670,400.122,177.370,26.726,154.380
C03188=1086.654,396.423,400.161,177.367,26.718,154.378
C03189=1086.648,396.176,400.200,177.364,26.710,154.377
C03190=1086.642,395.930,400.240,177.361,26.703,154.375
C03191=1086.636,395.684,400.279,177.357,26.695,154.374
C03192=1086.630,395.436,400.318,177.354,26.688,154.372
C03193=1086.624,395.189,400.358,177.351,26.680,154.371
C03194=1086.617,394.942,400.397,177.347,26.672,154.369
C03195=1086.611,394.696,400.436,177.343,26.665,154.368
C03196=1086.605,394.449,400.474,177.340,26.657,154.366
C03197=1086.598,394.202,400.514,177.337,26.649,154.365
C03198=1086.592,393.955,400.553,177.333,26.642,154.363
C03199=1086.586,393.709,400.592,177.330,26.634,154.362
C03200=1086.579,393.462,400.631,177.327,26.627,154.361
C03201=1086.573,393.215,400.670,177.323,26.619,154.359
C03202=1086.567,392.969,400.709,177.320,26.612,154.358
C03203=1086.561,392.721,400.747,177.317,26.605,154.356
C03204=1086.555,392.474,400.786,177.314,26.597,154.355
C03205=1086.549,392.228,400.825,177.310,26.590,154.353
C03206=1086.542,391.981,400.864,177.307,26.582,154.352
C03207=1086.535,391.734,400.903,177.304,26.575,154.351
C03208=1086.530,391.487,400.941,177.300,26.567,154.349
C03209=1086.523,391.240,400.980,177.297,26.560,154.348
C03210=1086.517,390.993,401.019,177.294,26.553,154.346
C03211=1086.510,390.747,401.057,177.290,26.546,154.345
C03212=1086.505,390.499,401.096,177.287,26.538,154.344
C03213=1086.498,390.253,401.135,177.284,26.531,154.342
C03214=1086.492,390.006,401.173,177.279,26.524,154.341
C03215=1086.485,389.759,401.212,177.276,26.517,154.340
C03216=1086.480,389.513,401.251,177.273,26.509,154.338
C03217=1086.473,389.265,401.289,177.269,26.502,154.337
C03218=1086.467,389.019,401.327,177.266,26.495,154.336
C03219=1086.460,388.772,401.365,177.263,26.488,154.334
C03220=1086.454,388.525,401.404,177.259,26.481,154.333
C03221=1086.448,388.278,401.443,177.257,26.474,154.332
C03222=1086.442,388.031,401.481,177.253,26.467,154.330
C03223=1086.436,387.784,401.519,177.250,26.460,154.329
C03224=1086.429,387.537,401.558,177.247,26.453,154.327
C03225=1086.423,387.291,401.596,177.243,26.446,154.326
C03226=1086.416,387.044,401.634,177.240,26.439,154.325
C03227=1086.411,386.797,401.673,177.237,26.432,154.324
C03228=1086.405,386.550,401.711,177.233,26.425,154.322
C03229=1086.398,386.303,401.749,177.230,26.418,154.321
C03230=1086.392,386.056,401.787,177.227,26.411,154.320
C03231=1086.386,385.809,401.825,177.223,26.404,154.318
C03232=1086.380,385.563,401.864,177.220,26.397,154.317
C03233=1086.373,385.315,401.902,177.216,26.390,154.316
C03234=1086.368,385.093,401.937,177.214,26.384,154.315
C03235=1086.362,384.871,401.970,177.210,26.377,154.313
C03236=1086.357,384.648,402.005,177.208,26.371,154.312
C03237=1086.352,384.426,402.040,177.204,26.365,154.311
C03238=1086.346,384.204,402.073,177.202,26.359,154.310
C03239=1086.341,383.981,402.108,177.199,26.353,154.309
C03240=1086.335,383.760,402.142,177.196,26.347,154.308
C03241=1086.330,383.537,402.175,177.193,26.341,154.307
C03242=1086.324,383.290,402.215,177.190,26.334,154.305
C03243=1086.318,383.043,402.252,177.186,26.327,154.304
C03244=1086.312,382.796,402.290,177.183,26.320,154.303
C03245=1086.306,382.550,402.328,177.179,26.313,154.302
C03246=1086.299,382.302,402.366,177.176,26.306,154.300
C03247=1086.293,382.056,402.403,177.173,26.300,154.299
C03248=1086.287,381.808,402.441,177.170,26.294,154.298
C03249=1086.281,381.561,402.478,177.167,26.287,154.297
C03250=1086.275,381.314,402.516,177.163,26.280,154.295
C03251=1086.268,381.067,402.554,177.160,26.274,154.294
C03252=1086.262,380.820,402.592,177.156,26.267,154.293
C03253=1086.256,380.574,402.629,177.153,26.260,154.292
C03254=1086.249,380.326,402.667,177.150,26.254,154.291
C03255=1086.244,380.079,402.704,177.147,26.248,154.290
C03256=1086.238,379.832,402.742,177.143,26.241,154.288
C03257=1086.232,379.585,402.780,177.140,26.235,154.287
C03258=1086.225,379.338,402.817,177.137,26.228,154.286
C03259=1086.219,379.091,402.854,177.133,26.222,154.285
C03260=1086.213,378.844,402.892,177.131,26.215,154.284
C03261=1086.207,378.597,402.930,177.127,26.209,154.282
C03262=1086.200,378.350,402.967,177.124,26.202,154.281
C03263=1086.194,378.103,403.004,177.120,26.196,154.280
C03264=1086.188,377.856,403.042,177.117,26.189,154.279
C03265=1086.183,377.609,403.079,177.114,26.183,154.278
C03266=1086.176,377.362,403.117,177.111,26.177,154.277
C03267=1086.170,377.114,403.154,177.107,26.170,154.275
C03268=1086.164,376.867,403.192,177.104,26.164,154.274
C03269=1086.157,376.621,403.229,177.101,26.158,154.273
C03270=1086.152,376.374,403.266,177.098,26.151,154.272
C03271=1086.146,376.126,403.303,177.095,26.145,154.271
C03272=1086.140,375.880,403.341,177.091,26.139,154.270
C03273=1086.133,375.632,403.377,177.089,26.132,154.269
C03274=1086.128,375.385,403.415,177.085,26.126,154.268
C03275=1086.122,375.138,403.452,177.082,26.120,154.266
C03276=1086.115,374.891,403.489,177.078,26.113,154.265
C03277=1086.110,374.644,403.526,177.076,26.107,154.264
C03278=1086.104,374.397,403.563,177.072,26.101,154.263
C03279=1086.097,374.150,403.601,177.069,26.095,154.262
C03280=1086.092,373.903,403.638,177.065,26.089,154.261
C03281=1086.086,373.656,403.674,177.063,26.082,154.260
C03282=1086.079,373.408,403.712,177.059,26.076,154.259
C03283=1086.073,373.161,403.749,177.056,26.070,154.258
C03284=1086.067,372.914,403.786,177.052,26.064,154.257
C03285=1086.061,372.667,403.822,177.049,26.058,154.256
C03286=1086.054,372.420,403.859,177.046,26.052,154.254
C03287=1086.049,372.172,403.896,177.042,26.046,154.253
C03288=1086.042,371.925,403.932,177.040,26.040,154.252
C03289=1086.037,371.679,403.970,177.036,26.034,154.251
C03290=1086.025,371.262,404.031,177.031,26.024,154.249
C03291=1086.015,370.845,404.093,177.025,26.014,154.248
C03292=1086.006,370.429,404.155,177.020,26.004,154.246
C03293=1085.995,370.012,404.218,177.014,25.993,154.244
C03294=1085.989,369.765,404.254,177.012,25.988,154.243
C03295=1085.982,369.518,404.290,177.008,25.982,154.242
C03296=1085.977,369.270,404.327,177.004,25.976,154.241
C03297=1085.971,369.023,404.363,177.002,25.970,154.240
C03298=1085.965,368.776,404.399,176.998,25.964,154.239
C03299=1085.959,368.529,404.436,176.995,25.958,154.238
C03300=1085.953,368.282,404.473,176.992,25.953,154.237
C03301=1085.947,368.035,404.509,176.989,25.946,154.236
C03302=1085.941,367.787,404.546,176.985,25.940,154.235
C03303=1085.935,367.540,404.582,176.983,25.935,154.234
C03304=1085.929,367.293,404.618,176.979,25.929,154.233
C03305=1085.923,367.045,404.655,176.976,25.923,154.232
C03306=1085.917,366.798,404.692,176.973,25.917,154.231
C03307=1085.911,366.551,404.728,176.969,25.911,154.230
C03308=1085.905,366.304,404.764,176.967,25.906,154.229
C03309=1085.900,366.057,404.801,176.963,25.900,154.228
C03310=1085.894,365.809,404.836,176.960,25.894,154.227
C03311=1085.887,365.562,404.873,176.957,25.888,154.226
C03312=1085.881,365.315,404.909,176.953,25.883,154.225
C03313=1085.875,365.067,404.945,176.950,25.877,154.224
C03314=1085.869,364.820,404.982,176.947,25.871,154.223
C03315=1085.863,364.572,405.018,176.944,25.866,154.222
C03316=1085.857,364.325,405.054,176.941,25.860,154.221
C03317=1085.851,364.078,405.090,176.937,25.854,154.220
C03318=1085.845,363.831,405.126,176.934,25.849,154.219
C03319=1085.839,363.584,405.162,176.931,25.843,154.218
C03320=1085.833,363.337,405.198,176.928,25.838,154.217
C03321=1085.827,363.089,405.234,176.925,25.832,154.216
C03322=1085.820,362.842,405.270,176.921,25.827,154.216
C03323=1085.815,362.595,405.306,176.918,25.821,154.214
C03324=1085.809,362.347,405.342,176.915,25.815,154.214
C03325=1085.803,362.100,405.378,176.912,25.810,154.213
C03326=1085.797,361.852,405.414,176.909,25.804,154.212
C03327=1085.791,361.605,405.449,176.905,25.799,154.211
C03328=1085.785,361.358,405.486,176.903,25.793,154.210
C03329=1085.779,361.111,405.521,176.899,25.788,154.209
C03330=1085.773,360.863,405.557,176.896,25.782,154.208
C03331=1085.766,360.616,405.593,176.893,25.777,154.207
C03332=1085.761,360.369,405.629,176.889,25.771,154.206
C03333=1085.755,360.121,405.665,176.886,25.766,154.205
C03334=1085.749,359.874,405.700,176.883,25.760,154.204
C03335=1085.743,359.626,405.736,176.880,25.755,154.203
C03336=1085.737,359.380,405.772,176.877,25.749,154.203
C03337=1085.730,359.132,405.807,176.874,25.744,154.202
C03338=1085.724,358.885,405.843,176.870,25.739,154.201
C03339=1085.718,358.637,405.879,176.867,25.734,154.200
C03340=1085.713,358.390,405.914,176.864,25.728,154.199
C03341=1085.707,358.142,405.950,176.861,25.723,154.198
C03342=1085.697,357.742,406.007,176.855,25.714,154.197
C03343=1085.687,357.340,406.065,176.851,25.705,154.195
C03344=1085.677,356.940,406.122,176.846,25.697,154.194
C03345=1085.668,356.539,406.179,176.840,25.688,154.192
C03346=1085.662,356.291,406.215,176.837,25.683,154.192
C03347=1085.656,356.044,406.250,176.834,25.677,154.191
C03348=1085.650,355.797,406.286,176.831,25.672,154.190
C03349=1085.644,355.550,406.321,176.827,25.667,154.189
C03350=1085.638,355.302,406.357,176.824,25.662,154.188
C03351=1085.632,355.054,406.392,176.821,25.656,154.187
C03352=1085.626,354.807,406.426,176.818,25.651,154.186
C03353=1085.620,354.559,406.462,176.815,25.646,154.186
C03354=1085.615,354.312,406.498,176.812,25.641,154.185
C03355=1085.608,354.065,406.533,176.809,25.636,154.184
C03356=1085.602,353.817,406.568,176.805,25.630,154.183
C03357=1085.597,353.570,406.603,176.803,25.625,154.182
C03358=1085.590,353.322,406.638,176.799,25.620,154.181
C03359=1085.585,353.075,406.674,176.796,25.615,154.181
C03360=1085.579,352.827,406.709,176.793,25.610,154.180
C03361=1085.573,352.580,406.743,176.790,25.605,154.179
C03362=1085.567,352.333,406.779,176.786,25.600,154.178
C03363=1085.560,352.085,406.813,176.784,25.594,154.177
C03364=1085.555,351.838,406.849,176.781,25.589,154.176
C03365=1085.548,351.590,406.883,176.777,25.584,154.176
C03366=1085.543,351.343,406.919,176.774,25.579,154.175
C03367=1085.536,351.096,406.954,176.771,25.574,154.174
C03368=1085.531,350.848,406.988,176.768,25.569,154.173
C03369=1085.524,350.601,407.024,176.764,25.564,154.172
C03370=1085.519,350.353,407.058,176.761,25.559,154.172
C03371=1085.512,350.106,407.093,176.759,25.554,154.171
C03372=1085.507,349.858,407.128,176.755,25.549,154.170
C03373=1085.501,349.610,407.162,176.752,25.544,154.169
C03374=1085.495,349.363,407.198,176.749,25.539,154.168
C03375=1085.489,349.115,407.232,176.746,25.534,154.168
C03376=1085.483,348.868,407.268,176.742,25.529,154.167
C03377=1085.477,348.620,407.302,176.739,25.524,154.166
C03378=1085.472,348.372,407.337,176.737,25.519,154.165
C03379=1085.465,348.125,407.372,176.733,25.514,154.164
C03380=1085.459,347.878,407.406,176.730,25.509,154.164
C03381=1085.454,347.630,407.440,176.727,25.504,154.163
C03382=1085.447,347.383,407.476,176.724,25.499,154.162
C03383=1085.441,347.136,407.510,176.721,25.494,154.161
C03384=1085.436,346.887,407.545,176.717,25.489,154.161
C03385=1085.430,346.640,407.579,176.715,25.484,154.160
C03386=1085.424,346.392,407.614,176.712,25.479,154.159
C03387=1085.418,346.145,407.648,176.708,25.475,154.158
C03388=1085.412,345.898,407.683,176.705,25.470,154.158
C03389=1085.406,345.649,407.718,176.702,25.465,154.157
C03390=1085.401,345.402,407.752,176.699,25.460,154.156
C03391=1085.395,345.155,407.786,176.696,25.455,154.155
C03392=1085.389,344.907,407.821,176.692,25.450,154.154
C03393=1085.383,344.659,407.855,176.690,25.445,154.154
C03394=1085.373,344.262,407.910,176.684,25.438,154.153
C03395=1085.364,343.863,407.966,176.680,25.430,154.151
C03396=1085.354,343.465,408.020,176.674,25.422,154.150
C03397=1085.344,343.068,408.075,176.669,25.414,154.149
C03398=1085.338,342.820,408.109,176.667,25.410,154.148
C03399=1085.333,342.572,408.144,176.663,25.405,154.148
C03400=1085.327,342.325,408.178,176.660,25.400,154.147
C03401=1085.321,342.078,408.212,176.657,25.396,154.146
C03402=1085.315,341.829,408.246,176.654,25.391,154.145
C03403=1085.309,341.582,408.280,176.651,25.386,154.145
C03404=1085.303,341.334,408.314,176.648,25.381,154.144
C03405=1085.297,341.086,408.349,176.645,25.377,154.143
C03406=1085.291,340.839,408.383,176.641,25.372,154.143
C03407=1085.285,340.592,408.417,176.639,25.367,154.142
C03408=1085.280,340.344,408.451,176.636,25.363,154.141
C03409=1085.274,340.096,408.485,176.632,25.358,154.140
C03410=1085.268,339.848,408.519,176.629,25.353,154.140
C03411=1085.262,339.601,408.553,176.626,25.349,154.139
C03412=1085.256,339.353,408.587,176.623,25.344,154.138
C03413=1085.250,339.106,408.621,176.620,25.339,154.137
C03414=1085.244,338.858,408.655,176.617,25.335,154.137
C03415=1085.238,338.610,408.688,176.614,25.330,154.136
C03416=1085.233,338.363,408.722,176.611,25.325,154.135
C03417=1085.227,338.115,408.756,176.608,25.321,154.135
C03418=1085.221,337.868,408.790,176.605,25.316,154.134
C03419=1085.215,337.620,408.824,176.601,25.311,154.133
C03420=1085.209,337.372,408.858,176.598,25.307,154.133
C03421=1085.203,337.124,408.892,176.595,25.303,154.132
C03422=1085.197,336.877,408.924,176.592,25.298,154.131
C03423=1085.191,336.629,408.958,176.589,25.293,154.131
C03424=1085.185,336.381,408.992,176.586,25.289,154.130
C03425=1085.179,336.134,409.026,176.583,25.284,154.129
C03426=1085.174,335.886,409.059,176.580,25.280,154.129
C03427=1085.168,335.638,409.094,176.576,25.275,154.128
C03428=1085.162,335.390,409.127,176.574,25.271,154.127
C03429=1085.156,335.144,409.160,176.571,25.266,154.127
C03430=1085.150,334.896,409.194,176.568,25.262,154.126
C03431=1085.144,334.648,409.228,176.564,25.257,154.125
C03432=1085.138,334.400,409.261,176.561,25.253,154.125
C03433=1085.132,334.152,409.295,176.558,25.248,154.124
C03434=1085.126,333.905,409.328,176.556,25.244,154.123
C03435=1085.120,333.657,409.362,176.553,25.240,154.123
C03436=1085.115,333.409,409.395,176.549,25.235,154.122
C03437=1085.109,333.162,409.429,176.546,25.230,154.121
C03438=1085.103,332.914,409.462,176.543,25.226,154.121
C03439=1085.097,332.666,409.495,176.540,25.221,154.120
C03440=1085.091,332.418,409.528,176.537,25.217,154.119
C03441=1085.086,332.170,409.562,176.534,25.212,154.119
C03442=1085.080,331.923,409.596,176.531,25.208,154.118
C03443=1085.074,331.676,409.629,176.528,25.204,154.117
C03444=1085.068,331.427,409.662,176.525,25.199,154.117
C03445=1085.061,331.179,409.695,176.521,25.195,154.116
C03446=1085.052,330.776,409.750,176.517,25.188,154.115
C03447=1085.042,330.372,409.803,176.512,25.181,154.114
C03448=1085.032,329.968,409.857,176.507,25.174,154.113
C03449=1085.023,329.564,409.911,176.502,25.167,154.112
C03450=1085.016,329.317,409.944,176.499,25.162,154.111
C03451=1085.011,329.069,409.977,176.496,25.159,154.111
C03452=1085.005,328.821,410.010,176.493,25.154,154.110
C03453=1084.999,328.573,410.043,176.489,25.150,154.110
C03454=1084.993,328.326,410.076,176.486,25.145,154.109
C03455=1084.987,328.078,410.109,176.484,25.141,154.108
C03456=1084.981,327.830,410.142,176.481,25.137,154.108
C03457=1084.975,327.582,410.175,176.478,25.132,154.107
C03458=1084.969,327.335,410.208,176.475,25.129,154.107
C03459=1084.963,327.087,410.241,176.472,25.124,154.106
C03460=1084.957,326.839,410.274,176.468,25.120,154.105
C03461=1084.951,326.592,410.307,176.465,25.115,154.105
C03462=1084.945,326.345,410.339,176.462,25.111,154.104
C03463=1084.940,326.096,410.372,176.459,25.107,154.104
C03464=1084.934,325.848,410.405,176.456,25.103,154.103
C03465=1084.928,325.601,410.438,176.454,25.099,154.103
C03466=1084.922,325.353,410.471,176.451,25.095,154.102
C03467=1084.916,325.105,410.503,176.447,25.090,154.101
C03468=1084.910,324.857,410.536,176.444,25.086,154.101
C03469=1084.904,324.609,410.569,176.441,25.082,154.100
C03470=1084.898,324.362,410.602,176.438,25.078,154.100
C03471=1084.892,324.113,410.634,176.435,25.073,154.099
C03472=1084.887,323.866,410.667,176.432,25.069,154.098
C03473=1084.881,323.618,410.700,176.429,25.065,154.098
C03474=1084.875,323.370,410.732,176.427,25.061,154.097
C03475=1084.869,323.123,410.765,176.423,25.057,154.097
C03476=1084.863,322.875,410.798,176.420,25.052,154.096
C03477=1084.857,322.626,410.830,176.417,25.048,154.095
C03478=1084.852,322.380,410.862,176.414,25.044,154.095
C03479=1084.846,322.131,410.895,176.411,25.040,154.094
C03480=1084.840,321.883,410.928,176.408,25.036,154.094
C03481=1084.834,321.635,410.960,176.405,25.031,154.093
C03482=1084.828,321.388,410.992,176.402,25.028,154.092
C03483=1084.823,321.140,411.025,176.399,25.024,154.092
C03484=1084.817,320.892,411.058,176.397,25.020,154.091
C03485=1084.811,320.644,411.090,176.393,25.015,154.091
C03486=1084.805,320.397,411.122,176.390,25.011,154.090
C03487=1084.800,320.149,411.155,176.387,25.007,154.090
C03488=1084.794,319.901,411.187,176.384,25.002,154.089
C03489=1084.788,319.653,411.219,176.381,24.998,154.088
C03490=1084.782,319.405,411.251,176.378,24.994,154.088
C03491=1084.777,319.157,411.284,176.375,24.990,154.087
C03492=1084.771,318.909,411.316,176.372,24.986,154.087
C03493=1084.765,318.662,411.349,176.369,24.982,154.086
C03494=1084.759,318.414,411.381,176.367,24.978,154.086
C03495=1084.754,318.166,411.413,176.364,24.974,154.085
C03496=1084.748,317.919,411.446,176.361,24.970,154.084
C03497=1084.742,317.670,411.478,176.358,24.966,154.084
C03498=1084.733,317.260,411.531,176.353,24.959,154.083
C03499=1084.723,316.849,411.585,176.347,24.952,154.082
C03500=1084.714,316.439,411.637,176.343,24.945,154.081
C03501=1084.704,316.029,411.691,176.338,24.939,154.080
C03502=1084.698,315.781,411.723,176.335,24.934,154.080
C03503=1084.694,315.533,411.755,176.332,24.930,154.079
C03504=1084.688,315.285,411.787,176.329,24.926,154.078
C03505=1084.682,315.037,411.819,176.326,24.922,154.078
C03506=1084.676,314.789,411.851,176.323,24.918,154.077
C03507=1084.670,314.541,411.883,176.321,24.914,154.077
C03508=1084.665,314.293,411.915,176.318,24.910,154.076
C03509=1084.658,314.045,411.946,176.315,24.906,154.076
C03510=1084.652,313.797,411.978,176.312,24.903,154.075
C03511=1084.646,313.549,412.010,176.309,24.899,154.075
C03512=1084.641,313.301,412.042,176.306,24.895,154.074
C03513=1084.634,313.054,412.073,176.303,24.891,154.074
C03514=1084.629,312.806,412.105,176.300,24.887,154.073
C03515=1084.623,312.558,412.137,176.296,24.883,154.073
C03516=1084.617,312.310,412.169,176.293,24.879,154.072
C03517=1084.611,312.062,412.200,176.290,24.875,154.072
C03518=1084.605,311.814,412.232,176.287,24.871,154.071
C03519=1084.599,311.567,412.264,176.284,24.867,154.071
C03520=1084.593,311.318,412.296,176.281,24.864,154.070
C03521=1084.587,311.071,412.327,176.278,24.860,154.070
C03522=1084.581,310.823,412.359,176.275,24.856,154.069
C03523=1084.575,310.575,412.391,176.272,24.852,154.069
C03524=1084.570,310.327,412.422,176.269,24.848,154.068
C03525=1084.563,310.079,412.453,176.266,24.844,154.068
C03526=1084.558,309.831,412.485,176.263,24.840,154.067
C03527=1084.552,309.583,412.517,176.260,24.836,154.067
C03528=1084.546,309.336,412.548,176.257,24.833,154.066
C03529=1084.540,309.087,412.579,176.254,24.829,154.066
C03530=1084.535,308.840,412.611,176.251,24.825,154.065
C03531=1084.528,308.592,412.642,176.249,24.821,154.065
C03532=1084.523,308.344,412.674,176.245,24.817,154.064
C03533=1084.517,308.095,412.705,176.243,24.814,154.064
C03534=1084.511,307.848,412.736,176.241,24.810,154.063
C03535=1084.505,307.600,412.768,176.237,24.806,154.063
C03536=1084.499,307.352,412.799,176.235,24.802,154.062
C03537=1084.494,307.105,412.830,176.232,24.798,154.062
C03538=1084.488,306.856,412.862,176.229,24.795,154.061
C03539=1084.482,306.608,412.893,176.226,24.791,154.061
C03540=1084.476,306.360,412.925,176.223,24.787,154.060
C03541=1084.471,306.112,412.956,176.220,24.783,154.060
C03542=1084.465,305.865,412.987,176.217,24.779,154.059
C03543=1084.459,305.616,413.018,176.214,24.775,154.059
C03544=1084.453,305.369,413.049,176.211,24.771,154.058
C03545=1084.448,305.121,413.081,176.208,24.768,154.058
C03546=1084.442,304.873,413.112,176.205,24.764,154.057
C03547=1084.436,304.625,413.142,176.202,24.760,154.057
C03548=1084.430,304.377,413.174,176.199,24.756,154.056
C03549=1084.424,304.129,413.205,176.196,24.752,154.056
C03550=1084.416,303.744,413.253,176.192,24.746,154.055
C03551=1084.407,303.359,413.302,176.187,24.741,154.054
C03552=1084.397,302.974,413.350,176.183,24.735,154.053
C03553=1084.389,302.589,413.398,176.177,24.728,154.053
C03554=1084.381,302.251,413.441,176.174,24.723,154.052
C03555=1084.376,302.003,413.472,176.171,24.719,154.051
C03556=1084.370,301.755,413.502,176.168,24.716,154.051
C03557=1084.364,301.508,413.534,176.165,24.712,154.051
C03558=1084.358,301.259,413.564,176.162,24.708,154.050
C03559=1084.353,301.011,413.595,176.159,24.704,154.050
C03560=1084.347,300.763,413.626,176.157,24.701,154.049
C03561=1084.342,300.516,413.657,176.154,24.697,154.049
C03562=1084.335,300.267,413.688,176.151,24.693,154.048
C03563=1084.330,300.019,413.719,176.148,24.690,154.048
C03564=1084.324,299.771,413.749,176.145,24.686,154.047
C03565=1084.319,299.523,413.780,176.142,24.682,154.047
C03566=1084.313,299.276,413.811,176.139,24.678,154.046
C03567=1084.308,299.027,413.843,176.136,24.674,154.046
C03568=1084.302,298.779,413.873,176.133,24.671,154.045
C03569=1084.296,298.531,413.903,176.130,24.667,154.045
C03570=1084.291,298.283,413.934,176.127,24.663,154.044
C03571=1084.285,298.035,413.965,176.125,24.659,154.044
C03572=1084.280,297.787,413.996,176.122,24.655,154.043
C03573=1084.274,297.539,414.026,176.119,24.652,154.043
C03574=1084.268,297.291,414.057,176.116,24.648,154.042
C03575=1084.262,297.043,414.087,176.113,24.644,154.042
C03576=1084.257,296.795,414.118,176.110,24.641,154.042
C03577=1084.251,296.547,414.148,176.107,24.637,154.041
C03578=1084.245,296.299,414.179,176.104,24.633,154.041
C03579=1084.239,296.051,414.209,176.101,24.630,154.040
C03580=1084.233,295.803,414.240,176.099,24.626,154.040
C03581=1084.228,295.555,414.271,176.096,24.623,154.039
C03582=1084.222,295.307,414.301,176.093,24.619,154.039
C03583=1084.216,295.059,414.331,176.090,24.615,154.038
C03584=1084.210,294.811,414.362,176.087,24.611,154.038
C03585=1084.204,294.563,414.392,176.084,24.608,154.037
C03586=1084.198,294.315,414.423,176.081,24.604,154.037
C03587=1084.193,294.067,414.452,176.079,24.601,154.036
C03588=1084.187,293.819,414.483,176.076,24.597,154.036
C03589=1084.181,293.571,414.513,176.073,24.594,154.036
C03590=1084.176,293.323,414.544,176.070,24.590,154.035
C03591=1084.170,293.075,414.574,176.067,24.586,154.035
C03592=1084.165,292.827,414.604,176.064,24.583,154.034
C03593=1084.158,292.578,414.635,176.061,24.579,154.034
C03594=1084.152,292.330,414.665,176.059,24.576,154.033
C03595=1084.147,292.082,414.696,176.056,24.572,154.033
C03596=1084.141,291.834,414.725,176.053,24.568,154.033
C03597=1084.135,291.586,414.756,176.050,24.564,154.032
C03598=1084.129,291.338,414.786,176.047,24.561,154.032
C03599=1084.124,291.090,414.816,176.044,24.557,154.031
C03600=1084.118,290.842,414.846,176.041,24.554,154.031
C03601=1084.112,290.594,414.876,176.039,24.550,154.030
C03602=1084.103,290.201,414.924,176.034,24.545,154.030
C03603=1084.094,289.807,414.972,176.029,24.539,154.029
C03604=1084.085,289.414,415.019,176.025,24.533,154.028
C03605=1084.076,289.020,415.067,176.020,24.528,154.028
C03606=1084.070,288.772,415.096,176.018,24.524,154.027
C03607=1084.064,288.524,415.127,176.015,24.521,154.027
C03608=1084.059,288.276,415.156,176.012,24.517,154.026
C03609=1084.053,288.028,415.187,176.009,24.513,154.026
C03610=1084.047,287.780,415.216,176.006,24.510,154.025
C03611=1084.041,287.532,415.246,176.003,24.506,154.025
C03612=1084.035,287.284,415.276,176.001,24.503,154.025
C03613=1084.029,287.036,415.306,175.998,24.500,154.024
C03614=1084.024,286.787,415.336,175.995,24.496,154.024
C03615=1084.018,286.539,415.365,175.992,24.493,154.023
C03616=1084.012,286.291,415.395,175.989,24.489,154.023
C03617=1084.006,286.043,415.425,175.987,24.485,154.023
C03618=1084.001,285.794,415.454,175.984,24.482,154.022
C03619=1083.995,285.547,415.485,175.981,24.478,154.022
C03620=1083.989,285.298,415.514,175.977,24.475,154.021
C03621=1083.983,285.050,415.543,175.974,24.471,154.021
C03622=1083.977,284.802,415.574,175.972,24.468,154.020
C03623=1083.972,284.554,415.603,175.969,24.464,154.020
C03624=1083.966,284.306,415.632,175.966,24.461,154.020
C03625=1083.961,284.058,415.662,175.963,24.457,154.019
C03626=1083.955,283.810,415.692,175.961,24.454,154.019
C03627=1083.949,283.562,415.722,175.958,24.450,154.018
C03628=1083.943,283.313,415.751,175.955,24.447,154.018
C03629=1083.938,283.065,415.780,175.952,24.443,154.018
C03630=1083.932,282.817,415.810,175.949,24.440,154.017
C03631=1083.926,282.569,415.840,175.947,24.436,154.017
C03632=1083.920,282.321,415.869,175.944,24.433,154.016
C03633=1083.915,282.073,415.899,175.941,24.429,154.016
C03634=1083.910,281.824,415.928,175.938,24.426,154.015
C03635=1083.903,281.576,415.957,175.936,24.423,154.015
C03636=1083.898,281.328,415.987,175.933,24.419,154.015
